LIN {X 0,Y 389.575,Z 385.776,A -85,B 0,C 180,E1 17407.486,E2 17407.486} C_VEL
LIN {X 0,Y 384.372,Z 564.348,A -85,B 0,C 180,E1 17404.221,E2 17404.221} C_VEL
LIN {X 0,Y 383.473,Z 583.113,A -85,B 0,C 180,E1 17403.623,E2 17403.623} C_VEL
LIN {X 0,Y 382.001,Z 600.901,A -85,B 0,C 180,E1 17402.806,E2 17402.806} C_VEL
LIN {X 0,Y 380.036,Z 618.183,A -85,B 0,C 180,E1 17401.748,E2 17401.748} C_VEL
LIN {X 0,Y 377.634,Z 634.674,A -85,B 0,C 180,E1 17400.465,E2 17400.465} C_VEL
LIN {X 0,Y 374.767,Z 651.083,A -85,B 0,C 180,E1 17398.874,E2 17398.874} C_VEL
LIN {X 0,Y 371.677,Z 666.384,A -85,B 0,C 180,E1 17397.04,E2 17397.04} C_VEL
LIN {X 0,Y 368.609,Z 680.089,A -85,B 0,C 180,E1 17395.033,E2 17395.033} C_VEL
LIN {X 0,Y 365.431,Z 693.192,A -85,B 0,C 180,E1 17392.692,E2 17392.692} C_VEL
LIN {X 0,Y 362.5,Z 704.69,A -85,B 0,C 180,E1 17390.168,E2 17390.168} C_VEL
LIN {X 0,Y 359.935,Z 714.65,A -85,B 0,C 180,E1 17387.458,E2 17387.458} C_VEL
LIN {X 0,Y 357.763,Z 723.094,A -85,B 0,C 180,E1 17384.568,E2 17384.568} C_VEL
LIN {X 0,Y 356.161,Z 729.667,A -85,B 0,C 180,E1 17381.661,E2 17381.661} C_VEL
LIN {X 0,Y 355.001,Z 734.817,A -85,B 0,C 180,E1 17378.585,E2 17378.585} C_VEL
LIN {X 0,Y 354.248,Z 738.439,A -85,B 0,C 180,E1 17375.344,E2 17375.344} C_VEL
LIN {X 0,Y 353.897,Z 740.346,A -85,B 0,C 180,E1 17372.105,E2 17372.105} C_VEL
LIN {X 0,Y 353.848,Z 740.616,A -85,B 0,C 180,E1 17368.867,E2 17368.867} C_VEL
LIN {X 0,Y 353.866,Z 740.566,A -85,B 0,C 180,E1 17368.451,E2 17368.451} C_VEL
LIN {X 0,Y 352.976,Z 740.398,A -85,B 0,C 180,E1 17367.201,E2 17367.201} C_VEL
LIN {X 0,Y 348.515,Z 739.641,A -85,B 0,C 180,E1 17364.746,E2 17364.746} C_VEL
LIN {X 0,Y 346.754,Z 738.536,A -85,B 0,C 180,E1 17363.218,E2 17363.218} C_VEL
LIN {X 0,Y 346.714,Z 738.05,A -85,B 0,C 180,E1 17362.764,E2 17362.764} C_VEL
LIN {X 0,Y 347.737,Z 733.66,A -85,B 0,C 180,E1 17359.537,E2 17359.537} C_VEL
LIN {X 0,Y 349.321,Z 727.307,A -85,B 0,C 180,E1 17356.257,E2 17356.257} C_VEL
LIN {X 0,Y 351.36,Z 719.697,A -85,B 0,C 180,E1 17353.297,E2 17353.297} C_VEL
LIN {X 0,Y 353.982,Z 710.063,A -85,B 0,C 180,E1 17350.36,E2 17350.36} C_VEL
LIN {X 0,Y 356.844,Z 699.482,A -85,B 0,C 180,E1 17347.775,E2 17347.775} C_VEL
LIN {X 0,Y 359.992,Z 687.464,A -85,B 0,C 180,E1 17345.38,E2 17345.38} C_VEL
LIN {X 0,Y 363.293,Z 673.927,A -85,B 0,C 180,E1 17343.17,E2 17343.17} C_VEL
LIN {X 0,Y 366.539,Z 659.329,A -85,B 0,C 180,E1 17341.22,E2 17341.22} C_VEL
LIN {X 0,Y 369.603,Z 643.731,A -85,B 0,C 180,E1 17339.522,E2 17339.522} C_VEL
LIN {X 0,Y 372.443,Z 626.719,A -85,B 0,C 180,E1 17338.031,E2 17338.031} C_VEL
LIN {X 0,Y 374.739,Z 609.542,A -85,B 0,C 180,E1 17336.842,E2 17336.842} C_VEL
LIN {X 0,Y 376.605,Z 590.744,A -85,B 0,C 180,E1 17335.852,E2 17335.852} C_VEL
LIN {X 0,Y 377.824,Z 571.243,A -85,B 0,C 180,E1 17335.127,E2 17335.127} C_VEL
LIN {X 0,Y 378.505,Z 547.045,A -85,B 0,C 180,E1 17334.58,E2 17334.58} C_VEL
LIN {X 0,Y 383.388,Z 388.518,A -85,B 0,C 180,E1 17331.66,E2 17331.66} C_VEL
LIN {X 0,Y 372.23,Z 368.985,A -85,B 0,C 180,E1 17329.629,E2 17329.629} C_VEL
LIN {X 0,Y 361.52,Z 352.259,A -85,B 0,C 180,E1 17327.541,E2 17327.541} C_VEL
LIN {X 0,Y 358.785,Z 347.938,A -85,B 0,C 180,E1 17326.899,E2 17326.899} C_VEL
LIN {X 0,Y 353.532,Z 335.825,A -85,B 0,C 180,E1 17323.861,E2 17323.861} C_VEL
LIN {X 0,Y 349.647,Z 327.602,A -85,B 0,C 180,E1 17321.563,E2 17321.563} C_VEL
LIN {X 0,Y 347.304,Z 322.978,A -85,B 0,C 180,E1 17320.157,E2 17320.157} C_VEL
LIN {X 0,Y 345.919,Z 319.541,A -85,B 0,C 180,E1 17319.059,E2 17319.059} C_VEL
LIN {X 0,Y 345.894,Z 319.384,A -85,B 0,C 180,E1 17314.823,E2 17314.823} C_VEL
LIN {X 0,Y 345.892,Z 319.382,A -85,B 0,C 180,E1 17310.527,E2 17310.527} C_VEL
LIN {X 0,Y 345.896,Z 319.388,A -85,B 0,C 180,E1 17306.354,E2 17306.354} C_VEL
LIN {X 0,Y 345.893,Z 319.4,A -85,B 0,C 180,E1 17302.252,E2 17302.252} C_VEL
LIN {X 0,Y 345.899,Z 319.385,A -85,B 0,C 180,E1 17298.014,E2 17298.014} C_VEL
LIN {X 0,Y 345.906,Z 319.366,A -85,B 0,C 180,E1 17293.785,E2 17293.785} C_VEL
LIN {X 0,Y 345.898,Z 319.37,A -85,B 0,C 180,E1 17289.484,E2 17289.484} C_VEL
LIN {X 0,Y 345.89,Z 319.398,A -85,B 0,C 180,E1 17285.308,E2 17285.308} C_VEL
LIN {X 0,Y 345.877,Z 319.386,A -85,B 0,C 180,E1 17281.16,E2 17281.16} C_VEL
LIN {X 0,Y 345.871,Z 319.369,A -85,B 0,C 180,E1 17277.018,E2 17277.018} C_VEL
LIN {X 0,Y 345.87,Z 319.378,A -85,B 0,C 180,E1 17272.86,E2 17272.86} C_VEL
LIN {X 0,Y 345.873,Z 319.401,A -85,B 0,C 180,E1 17268.664,E2 17268.664} C_VEL
LIN {X 0,Y 345.873,Z 319.4,A -85,B 0,C 180,E1 17264.405,E2 17264.405} C_VEL
LIN {X 0,Y 345.88,Z 319.39,A -85,B 0,C 180,E1 17260.056,E2 17260.056} C_VEL
LIN {X 0,Y 345.886,Z 319.384,A -85,B 0,C 180,E1 17255.947,E2 17255.947} C_VEL
LIN {X 0,Y 345.901,Z 319.385,A -85,B 0,C 180,E1 17251.702,E2 17251.702} C_VEL
LIN {X 0,Y 345.947,Z 319.628,A -85,B 0,C 180,E1 17249.507,E2 17249.507} C_VEL
LIN {X 0,Y 347.584,Z 323.392,A -85,B 0,C 180,E1 17248.43,E2 17248.43} C_VEL
LIN {X 0,Y 348.628,Z 324.913,A -85,B 0,C 180,E1 17247.956,E2 17247.956} C_VEL
LIN {X 0,Y 353.831,Z 334.918,A -85,B 0,C 180,E1 17245.39,E2 17245.39} C_VEL
LIN {X 0,Y 357.949,Z 342.981,A -85,B 0,C 180,E1 17243.49,E2 17243.49} C_VEL
LIN {X 0,Y 364.694,Z 357.152,A -85,B 0,C 180,E1 17240.502,E2 17240.502} C_VEL
LIN {X 0,Y 371.956,Z 374.258,A -85,B 0,C 180,E1 17237.359,E2 17237.359} C_VEL
LIN {X 0,Y 374.056,Z 379.335,A -85,B 0,C 180,E1 17236.557,E2 17236.557} C_VEL
LIN {X 0,Y 381.034,Z 392.431,A -85,B 0,C 180,E1 17235.246,E2 17235.246} C_VEL
LIN {X 0,Y 383.985,Z 429.126,A -85,B 0,C 180,E1 17233.918,E2 17233.918} C_VEL
LIN {X 0,Y 375.667,Z 632.493,A -85,B 0,C 180,E1 17229.71,E2 17229.71} C_VEL
LIN {X 0,Y 373.709,Z 654.478,A -85,B 0,C 180,E1 17229.004,E2 17229.004} C_VEL
LIN {X 0,Y 371.041,Z 675.386,A -85,B 0,C 180,E1 17228.054,E2 17228.054} C_VEL
LIN {X 0,Y 368.083,Z 694.62,A -85,B 0,C 180,E1 17226.892,E2 17226.892} C_VEL
LIN {X 0,Y 364.802,Z 713.742,A -85,B 0,C 180,E1 17225.427,E2 17225.427} C_VEL
LIN {X 0,Y 361.389,Z 732.08,A -85,B 0,C 180,E1 17223.691,E2 17223.691} C_VEL
LIN {X 0,Y 357.817,Z 750.227,A -85,B 0,C 180,E1 17221.596,E2 17221.596} C_VEL
LIN {X 0,Y 354.467,Z 767.276,A -85,B 0,C 180,E1 17219.207,E2 17219.207} C_VEL
LIN {X 0,Y 351.414,Z 783.149,A -85,B 0,C 180,E1 17216.531,E2 17216.531} C_VEL
LIN {X 0,Y 348.903,Z 797.366,A -85,B 0,C 180,E1 17213.653,E2 17213.653} C_VEL
LIN {X 0,Y 346.99,Z 809.978,A -85,B 0,C 180,E1 17210.581,E2 17210.581} C_VEL
LIN {X 0,Y 345.729,Z 820.44,A -85,B 0,C 180,E1 17207.503,E2 17207.503} C_VEL
LIN {X 0,Y 345.044,Z 829.017,A -85,B 0,C 180,E1 17204.43,E2 17204.43} C_VEL
LIN {X 0,Y 344.787,Z 836.104,A -85,B 0,C 180,E1 17201.203,E2 17201.203} C_VEL
LIN {X 0,Y 344.85,Z 841.123,A -85,B 0,C 180,E1 17198.167,E2 17198.167} C_VEL
LIN {X 0,Y 345.058,Z 844.743,A -85,B 0,C 180,E1 17194.987,E2 17194.987} C_VEL
LIN {X 0,Y 345.211,Z 846.508,A -85,B 0,C 180,E1 17192.158,E2 17192.158} C_VEL
LIN {X 0,Y 345.255,Z 846.827,A -85,B 0,C 180,E1 17189.17,E2 17189.17} C_VEL
LIN {X 0,Y 345.126,Z 845.656,A -85,B 0,C 180,E1 17186.179,E2 17186.179} C_VEL
LIN {X 0,Y 344.931,Z 842.863,A -85,B 0,C 180,E1 17183.175,E2 17183.175} C_VEL
LIN {X 0,Y 344.793,Z 838.223,A -85,B 0,C 180,E1 17179.98,E2 17179.98} C_VEL
LIN {X 0,Y 344.896,Z 831.799,A -85,B 0,C 180,E1 17176.761,E2 17176.761} C_VEL
LIN {X 0,Y 345.408,Z 823.997,A -85,B 0,C 180,E1 17173.693,E2 17173.693} C_VEL
LIN {X 0,Y 346.494,Z 813.722,A -85,B 0,C 180,E1 17170.444,E2 17170.444} C_VEL
LIN {X 0,Y 348.173,Z 801.841,A -85,B 0,C 180,E1 17167.369,E2 17167.369} C_VEL
LIN {X 0,Y 350.447,Z 788.441,A -85,B 0,C 180,E1 17164.481,E2 17164.481} C_VEL
LIN {X 0,Y 353.14,Z 774.009,A -85,B 0,C 180,E1 17161.874,E2 17161.874} C_VEL
LIN {X 0,Y 356.244,Z 758.161,A -85,B 0,C 180,E1 17159.47,E2 17159.47} C_VEL
LIN {X 0,Y 359.673,Z 740.767,A -85,B 0,C 180,E1 17157.27,E2 17157.27} C_VEL
LIN {X 0,Y 363.194,Z 722.371,A -85,B 0,C 180,E1 17155.356,E2 17155.356} C_VEL
LIN {X 0,Y 366.647,Z 702.966,A -85,B 0,C 180,E1 17153.719,E2 17153.719} C_VEL
LIN {X 0,Y 369.743,Z 683.735,A -85,B 0,C 180,E1 17152.426,E2 17152.426} C_VEL
LIN {X 0,Y 372.564,Z 663.659,A -85,B 0,C 180,E1 17151.389,E2 17151.389} C_VEL
LIN {X 0,Y 374.836,Z 642.783,A -85,B 0,C 180,E1 17150.598,E2 17150.598} C_VEL
LIN {X 0,Y 376.217,Z 620.758,A -85,B 0,C 180,E1 17150.027,E2 17150.027} C_VEL
LIN {X 0,Y 383.944,Z 427.198,A -85,B 0,C 180,E1 17146.047,E2 17146.047} C_VEL
LIN {X 0,Y 380.702,Z 391.532,A -85,B 0,C 180,E1 17144.711,E2 17144.711} C_VEL
LIN {X 0,Y 373.38,Z 377.914,A -85,B 0,C 180,E1 17143.277,E2 17143.277} C_VEL
LIN {X 0,Y 366.854,Z 362.006,A -85,B 0,C 180,E1 17140.441,E2 17140.441} C_VEL
LIN {X 0,Y 360.67,Z 348.666,A -85,B 0,C 180,E1 17137.782,E2 17137.782} C_VEL
LIN {X 0,Y 355.146,Z 337.373,A -85,B 0,C 180,E1 17135.25,E2 17135.25} C_VEL
LIN {X 0,Y 350.284,Z 328.233,A -85,B 0,C 180,E1 17132.947,E2 17132.947} C_VEL
LIN {X 0,Y 348.264,Z 324.159,A -85,B 0,C 180,E1 17131.888,E2 17131.888} C_VEL
LIN {X 0,Y 346.287,Z 320.952,A -85,B 0,C 180,E1 17130.927,E2 17130.927} C_VEL
LIN {X 0,Y 345.918,Z 319.456,A -85,B 0,C 180,E1 17130.413,E2 17130.413} C_VEL
LIN {X 0,Y 345.898,Z 319.385,A -85,B 0,C 180,E1 17126.248,E2 17126.248} C_VEL
LIN {X 0,Y 345.886,Z 319.383,A -85,B 0,C 180,E1 17122.073,E2 17122.073} C_VEL
LIN {X 0,Y 345.877,Z 319.378,A -85,B 0,C 180,E1 17117.844,E2 17117.844} C_VEL
LIN {X 0,Y 345.87,Z 319.372,A -85,B 0,C 180,E1 17113.542,E2 17113.542} C_VEL
LIN {X 0,Y 345.87,Z 319.379,A -85,B 0,C 180,E1 17109.316,E2 17109.316} C_VEL
LIN {X 0,Y 345.873,Z 319.402,A -85,B 0,C 180,E1 17105.141,E2 17105.141} C_VEL
LIN {X 0,Y 345.872,Z 319.39,A -85,B 0,C 180,E1 17100.993,E2 17100.993} C_VEL
LIN {X 0,Y 345.87,Z 319.369,A -85,B 0,C 180,E1 17096.851,E2 17096.851} C_VEL
LIN {X 0,Y 345.884,Z 319.379,A -85,B 0,C 180,E1 17092.692,E2 17092.692} C_VEL
LIN {X 0,Y 345.897,Z 319.401,A -85,B 0,C 180,E1 17088.491,E2 17088.491} C_VEL
LIN {X 0,Y 345.908,Z 319.379,A -85,B 0,C 180,E1 17084.234,E2 17084.234} C_VEL
LIN {X 0,Y 345.896,Z 319.37,A -85,B 0,C 180,E1 17079.956,E2 17079.956} C_VEL
LIN {X 0,Y 345.902,Z 319.373,A -85,B 0,C 180,E1 17075.947,E2 17075.947} C_VEL
LIN {X 0,Y 345.896,Z 319.385,A -85,B 0,C 180,E1 17071.701,E2 17071.701} C_VEL
LIN {X 0,Y 345.897,Z 319.393,A -85,B 0,C 180,E1 17067.569,E2 17067.569} C_VEL
LIN {X 0,Y 345.896,Z 319.393,A -85,B 0,C 180,E1 17063.453,E2 17063.453} C_VEL
LIN {X 0,Y 345.937,Z 319.68,A -85,B 0,C 180,E1 17060.73,E2 17060.73} C_VEL
LIN {X 0,Y 347.422,Z 323.162,A -85,B 0,C 180,E1 17059.643,E2 17059.643} C_VEL
LIN {X 0,Y 348.545,Z 325.55,A -85,B 0,C 180,E1 17058.934,E2 17058.934} C_VEL
LIN {X 0,Y 350.596,Z 329.771,A -85,B 0,C 180,E1 17057.697,E2 17057.697} C_VEL
LIN {X 0,Y 354.243,Z 337.521,A -85,B 0,C 180,E1 17055.568,E2 17055.568} C_VEL
LIN {X 0,Y 358.954,Z 348.373,A -85,B 0,C 180,E1 17052.896,E2 17052.896} C_VEL
LIN {X 0,Y 369.652,Z 364.898,A -85,B 0,C 180,E1 17050.738,E2 17050.738} C_VEL
LIN {X 0,Y 379.94,Z 382.361,A -85,B 0,C 180,E1 17048.834,E2 17048.834} C_VEL
LIN {X 0,Y 383.444,Z 389.074,A -85,B 0,C 180,E1 17048.206,E2 17048.206} C_VEL
LIN {X 0,Y 378.018,Z 564.942,A -85,B 0,C 180,E1 17044.946,E2 17044.946} C_VEL
LIN {X 0,Y 377.086,Z 583.644,A -85,B 0,C 180,E1 17044.345,E2 17044.345} C_VEL
LIN {X 0,Y 375.513,Z 601.927,A -85,B 0,C 180,E1 17043.496,E2 17043.496} C_VEL
LIN {X 0,Y 373.525,Z 618.693,A -85,B 0,C 180,E1 17042.458,E2 17042.458} C_VEL
LIN {X 0,Y 370.899,Z 636.019,A -85,B 0,C 180,E1 17041.094,E2 17041.094} C_VEL
LIN {X 0,Y 367.89,Z 652.482,A -85,B 0,C 180,E1 17039.466,E2 17039.466} C_VEL
LIN {X 0,Y 364.669,Z 667.723,A -85,B 0,C 180,E1 17037.604,E2 17037.604} C_VEL
LIN {X 0,Y 361.466,Z 681.388,A -85,B 0,C 180,E1 17035.563,E2 17035.563} C_VEL
LIN {X 0,Y 358.145,Z 694.464,A -85,B 0,C 180,E1 17033.18,E2 17033.18} C_VEL
LIN {X 0,Y 355.074,Z 705.939,A -85,B 0,C 180,E1 17030.608,E2 17030.608} C_VEL
LIN {X 0,Y 352.38,Z 715.885,A -85,B 0,C 180,E1 17027.845,E2 17027.845} C_VEL
LIN {X 0,Y 350.093,Z 724.318,A -85,B 0,C 180,E1 17024.894,E2 17024.894} C_VEL
LIN {X 0,Y 348.354,Z 731.066,A -85,B 0,C 180,E1 17021.831,E2 17021.831} C_VEL
LIN {X 0,Y 347.117,Z 736.256,A -85,B 0,C 180,E1 17018.614,E2 17018.614} C_VEL
LIN {X 0,Y 346.367,Z 739.644,A -85,B 0,C 180,E1 17015.466,E2 17015.466} C_VEL
LIN {X 0,Y 345.992,Z 741.548,A -85,B 0,C 180,E1 17012.153,E2 17012.153} C_VEL
LIN {X 0,Y 345.939,Z 741.818,A -85,B 0,C 180,E1 17008.841,E2 17008.841} C_VEL
LIN {X 0,Y 346.204,Z 740.465,A -85,B 0,C 180,E1 17005.528,E2 17005.528} C_VEL
LIN {X 0,Y 346.714,Z 738.05,A -85,B 0,C 180,E1 17002.764,E2 17002.764} C_VEL
LIN {X 0,Y 346.061,Z 736.752,A -85,B 0,C 180,E1 17001.504,E2 17001.504} C_VEL
LIN {X 0,Y 341.253,Z 732.89,A -85,B 0,C 180,E1 16998.207,E2 16998.207} C_VEL
LIN {X 0,Y 340.994,Z 730.849,A -85,B 0,C 180,E1 16997.039,E2 16997.039} C_VEL
LIN {X 0,Y 342.986,Z 723.691,A -85,B 0,C 180,E1 16993.923,E2 16993.923} C_VEL
LIN {X 0,Y 345.546,Z 714.785,A -85,B 0,C 180,E1 16990.916,E2 16990.916} C_VEL
LIN {X 0,Y 348.539,Z 704.306,A -85,B 0,C 180,E1 16988.104,E2 16988.104} C_VEL
LIN {X 0,Y 351.909,Z 692.224,A -85,B 0,C 180,E1 16985.493,E2 16985.493} C_VEL
LIN {X 0,Y 355.499,Z 678.411,A -85,B 0,C 180,E1 16983.076,E2 16983.076} C_VEL
LIN {X 0,Y 358.999,Z 663.723,A -85,B 0,C 180,E1 16980.99,E2 16980.99} C_VEL
LIN {X 0,Y 362.256,Z 648.294,A -85,B 0,C 180,E1 16979.204,E2 16979.204} C_VEL
LIN {X 0,Y 365.281,Z 631.623,A -85,B 0,C 180,E1 16977.648,E2 16977.648} C_VEL
LIN {X 0,Y 367.892,Z 613.759,A -85,B 0,C 180,E1 16976.33,E2 16976.33} C_VEL
LIN {X 0,Y 369.927,Z 595.416,A -85,B 0,C 180,E1 16975.295,E2 16975.295} C_VEL
LIN {X 0,Y 371.317,Z 576.435,A -85,B 0,C 180,E1 16974.519,E2 16974.519} C_VEL
LIN {X 0,Y 372.031,Z 556.598,A -85,B 0,C 180,E1 16973.998,E2 16973.998} C_VEL
LIN {X 0,Y 377.33,Z 391.658,A -85,B 0,C 180,E1 16970.912,E2 16970.912} C_VEL
LIN {X 0,Y 366.892,Z 373.263,A -85,B 0,C 180,E1 16968.936,E2 16968.936} C_VEL
LIN {X 0,Y 356.62,Z 357.168,A -85,B 0,C 180,E1 16966.859,E2 16966.859} C_VEL
LIN {X 0,Y 351.137,Z 348.844,A -85,B 0,C 180,E1 16965.621,E2 16965.621} C_VEL
LIN {X 0,Y 345.873,Z 337.173,A -85,B 0,C 180,E1 16962.512,E2 16962.512} C_VEL
LIN {X 0,Y 341.765,Z 328.63,A -85,B 0,C 180,E1 16959.961,E2 16959.961} C_VEL
LIN {X 0,Y 339.688,Z 324.424,A -85,B 0,C 180,E1 16958.61,E2 16958.61} C_VEL
LIN {X 0,Y 337.986,Z 320.54,A -85,B 0,C 180,E1 16957.273,E2 16957.273} C_VEL
LIN {X 0,Y 337.951,Z 320.371,A -85,B 0,C 180,E1 16952.983,E2 16952.983} C_VEL
LIN {X 0,Y 337.95,Z 320.368,A -85,B 0,C 180,E1 16948.64,E2 16948.64} C_VEL
LIN {X 0,Y 337.952,Z 320.361,A -85,B 0,C 180,E1 16944.326,E2 16944.326} C_VEL
LIN {X 0,Y 337.949,Z 320.361,A -85,B 0,C 180,E1 16940.253,E2 16940.253} C_VEL
LIN {X 0,Y 337.96,Z 320.373,A -85,B 0,C 180,E1 16935.953,E2 16935.953} C_VEL
LIN {X 0,Y 337.964,Z 320.385,A -85,B 0,C 180,E1 16931.699,E2 16931.699} C_VEL
LIN {X 0,Y 337.964,Z 320.361,A -85,B 0,C 180,E1 16927.48,E2 16927.48} C_VEL
LIN {X 0,Y 337.939,Z 320.356,A -85,B 0,C 180,E1 16923.223,E2 16923.223} C_VEL
LIN {X 0,Y 337.929,Z 320.376,A -85,B 0,C 180,E1 16918.983,E2 16918.983} C_VEL
LIN {X 0,Y 337.927,Z 320.39,A -85,B 0,C 180,E1 16914.738,E2 16914.738} C_VEL
LIN {X 0,Y 337.926,Z 320.37,A -85,B 0,C 180,E1 16910.463,E2 16910.463} C_VEL
LIN {X 0,Y 337.932,Z 320.361,A -85,B 0,C 180,E1 16906.134,E2 16906.134} C_VEL
LIN {X 0,Y 337.943,Z 320.364,A -85,B 0,C 180,E1 16901.901,E2 16901.901} C_VEL
LIN {X 0,Y 337.955,Z 320.368,A -85,B 0,C 180,E1 16897.748,E2 16897.748} C_VEL
LIN {X 0,Y 337.969,Z 320.367,A -85,B 0,C 180,E1 16893.467,E2 16893.467} C_VEL
LIN {X 0,Y 338.026,Z 320.649,A -85,B 0,C 180,E1 16891.307,E2 16891.307} C_VEL
LIN {X 0,Y 339.317,Z 323.956,A -85,B 0,C 180,E1 16890.328,E2 16890.328} C_VEL
LIN {X 0,Y 340.859,Z 326.12,A -85,B 0,C 180,E1 16889.585,E2 16889.585} C_VEL
LIN {X 0,Y 342.798,Z 329.791,A -85,B 0,C 180,E1 16888.527,E2 16888.527} C_VEL
LIN {X 0,Y 348.279,Z 340.218,A -85,B 0,C 180,E1 16885.758,E2 16885.758} C_VEL
LIN {X 0,Y 354.382,Z 352.579,A -85,B 0,C 180,E1 16882.859,E2 16882.859} C_VEL
LIN {X 0,Y 360.708,Z 366.49,A -85,B 0,C 180,E1 16879.978,E2 16879.978} C_VEL
LIN {X 0,Y 365.81,Z 378.592,A -85,B 0,C 180,E1 16877.802,E2 16877.802} C_VEL
LIN {X 0,Y 375.242,Z 395.721,A -85,B 0,C 180,E1 16875.957,E2 16875.957} C_VEL
LIN {X 0,Y 377.885,Z 430.233,A -85,B 0,C 180,E1 16874.686,E2 16874.686} C_VEL
LIN {X 0,Y 369.297,Z 631.618,A -85,B 0,C 180,E1 16870.468,E2 16870.468} C_VEL
LIN {X 0,Y 367.272,Z 653.63,A -85,B 0,C 180,E1 16869.753,E2 16869.753} C_VEL
LIN {X 0,Y 364.435,Z 674.971,A -85,B 0,C 180,E1 16868.771,E2 16868.771} C_VEL
LIN {X 0,Y 361.176,Z 695.239,A -85,B 0,C 180,E1 16867.518,E2 16867.518} C_VEL
LIN {X 0,Y 357.602,Z 714.966,A -85,B 0,C 180,E1 16865.955,E2 16865.955} C_VEL
LIN {X 0,Y 353.991,Z 733.289,A -85,B 0,C 180,E1 16864.149,E2 16864.149} C_VEL
LIN {X 0,Y 350.491,Z 750.079,A -85,B 0,C 180,E1 16862.142,E2 16862.142} C_VEL
LIN {X 0,Y 347.071,Z 766.57,A -85,B 0,C 180,E1 16859.772,E2 16859.772} C_VEL
LIN {X 0,Y 343.961,Z 781.792,A -85,B 0,C 180,E1 16857.153,E2 16857.153} C_VEL
LIN {X 0,Y 341.276,Z 796.036,A -85,B 0,C 180,E1 16854.215,E2 16854.215} C_VEL
LIN {X 0,Y 339.307,Z 808.039,A -85,B 0,C 180,E1 16851.25,E2 16851.25} C_VEL
LIN {X 0,Y 337.908,Z 818.643,A -85,B 0,C 180,E1 16848.1,E2 16848.1} C_VEL
LIN {X 0,Y 337.111,Z 827.752,A -85,B 0,C 180,E1 16844.777,E2 16844.777} C_VEL
LIN {X 0,Y 336.824,Z 834.857,A -85,B 0,C 180,E1 16841.472,E2 16841.472} C_VEL
LIN {X 0,Y 336.893,Z 839.896,A -85,B 0,C 180,E1 16838.362,E2 16838.362} C_VEL
LIN {X 0,Y 337.125,Z 843.531,A -85,B 0,C 180,E1 16835.104,E2 16835.104} C_VEL
LIN {X 0,Y 337.296,Z 845.304,A -85,B 0,C 180,E1 16832.208,E2 16832.208} C_VEL
LIN {X 0,Y 337.344,Z 845.625,A -85,B 0,C 180,E1 16829.151,E2 16829.151} C_VEL
LIN {X 0,Y 337.2,Z 844.447,A -85,B 0,C 180,E1 16826.09,E2 16826.09} C_VEL
LIN {X 0,Y 336.979,Z 841.641,A -85,B 0,C 180,E1 16823.013,E2 16823.013} C_VEL
LIN {X 0,Y 336.832,Z 836.984,A -85,B 0,C 180,E1 16819.741,E2 16819.741} C_VEL
LIN {X 0,Y 336.947,Z 830.538,A -85,B 0,C 180,E1 16816.443,E2 16816.443} C_VEL
LIN {X 0,Y 337.497,Z 822.711,A -85,B 0,C 180,E1 16813.3,E2 16813.3} C_VEL
LIN {X 0,Y 338.683,Z 812.419,A -85,B 0,C 180,E1 16809.974,E2 16809.974} C_VEL
LIN {X 0,Y 340.528,Z 800.34,A -85,B 0,C 180,E1 16806.784,E2 16806.784} C_VEL
LIN {X 0,Y 342.929,Z 787.093,A -85,B 0,C 180,E1 16803.88,E2 16803.88} C_VEL
LIN {X 0,Y 345.7,Z 773.129,A -85,B 0,C 180,E1 16801.308,E2 16801.308} C_VEL
LIN {X 0,Y 348.97,Z 757.336,A -85,B 0,C 180,E1 16798.859,E2 16798.859} C_VEL
LIN {X 0,Y 352.569,Z 740.004,A -85,B 0,C 180,E1 16796.622,E2 16796.622} C_VEL
LIN {X 0,Y 356.261,Z 721.682,A -85,B 0,C 180,E1 16794.681,E2 16794.681} C_VEL
LIN {X 0,Y 359.684,Z 703.397,A -85,B 0,C 180,E1 16793.1,E2 16793.1} C_VEL
LIN {X 0,Y 362.893,Z 684.551,A -85,B 0,C 180,E1 16791.791,E2 16791.791} C_VEL
LIN {X 0,Y 365.952,Z 663.876,A -85,B 0,C 180,E1 16790.69,E2 16790.69} C_VEL
LIN {X 0,Y 368.407,Z 642.256,A -85,B 0,C 180,E1 16789.855,E2 16789.855} C_VEL
LIN {X 0,Y 369.854,Z 620.163,A -85,B 0,C 180,E1 16789.272,E2 16789.272} C_VEL
LIN {X 0,Y 377.84,Z 428.2,A -85,B 0,C 180,E1 16785.277,E2 16785.277} C_VEL
LIN {X 0,Y 374.987,Z 395.198,A -85,B 0,C 180,E1 16784.021,E2 16784.021} C_VEL
LIN {X 0,Y 365.339,Z 377.727,A -85,B 0,C 180,E1 16782.106,E2 16782.106} C_VEL
LIN {X 0,Y 358.592,Z 361.64,A -85,B 0,C 180,E1 16779.061,E2 16779.061} C_VEL
LIN {X 0,Y 351.937,Z 347.377,A -85,B 0,C 180,E1 16776.021,E2 16776.021} C_VEL
LIN {X 0,Y 346.773,Z 337.483,A -85,B 0,C 180,E1 16773.565,E2 16773.565} C_VEL
LIN {X 0,Y 344.569,Z 333.342,A -85,B 0,C 180,E1 16772.468,E2 16772.468} C_VEL
LIN {X 0,Y 342.71,Z 329.695,A -85,B 0,C 180,E1 16771.482,E2 16771.482} C_VEL
LIN {X 0,Y 340.761,Z 325.802,A -85,B 0,C 180,E1 16770.387,E2 16770.387} C_VEL
LIN {X 0,Y 338.388,Z 322.126,A -85,B 0,C 180,E1 16769.178,E2 16769.178} C_VEL
LIN {X 0,Y 338,Z 320.488,A -85,B 0,C 180,E1 16768.634,E2 16768.634} C_VEL
LIN {X 0,Y 337.962,Z 320.376,A -85,B 0,C 180,E1 16764.33,E2 16764.33} C_VEL
LIN {X 0,Y 337.957,Z 320.383,A -85,B 0,C 180,E1 16760.252,E2 16760.252} C_VEL
LIN {X 0,Y 337.942,Z 320.391,A -85,B 0,C 180,E1 16755.942,E2 16755.942} C_VEL
LIN {X 0,Y 337.932,Z 320.383,A -85,B 0,C 180,E1 16751.607,E2 16751.607} C_VEL
LIN {X 0,Y 337.928,Z 320.366,A -85,B 0,C 180,E1 16747.309,E2 16747.309} C_VEL
LIN {X 0,Y 337.93,Z 320.359,A -85,B 0,C 180,E1 16743.053,E2 16743.053} C_VEL
LIN {X 0,Y 337.931,Z 320.38,A -85,B 0,C 180,E1 16738.982,E2 16738.982} C_VEL
LIN {X 0,Y 337.943,Z 320.386,A -85,B 0,C 180,E1 16734.737,E2 16734.737} C_VEL
LIN {X 0,Y 337.954,Z 320.359,A -85,B 0,C 180,E1 16730.463,E2 16730.463} C_VEL
LIN {X 0,Y 337.957,Z 320.356,A -85,B 0,C 180,E1 16726.134,E2 16726.134} C_VEL
LIN {X 0,Y 337.951,Z 320.374,A -85,B 0,C 180,E1 16721.901,E2 16721.901} C_VEL
LIN {X 0,Y 337.951,Z 320.389,A -85,B 0,C 180,E1 16717.746,E2 16717.746} C_VEL
LIN {X 0,Y 337.946,Z 320.38,A -85,B 0,C 180,E1 16713.464,E2 16713.464} C_VEL
LIN {X 0,Y 337.945,Z 320.375,A -85,B 0,C 180,E1 16709.213,E2 16709.213} C_VEL
LIN {X 0,Y 337.949,Z 320.375,A -85,B 0,C 180,E1 16704.972,E2 16704.972} C_VEL
LIN {X 0,Y 338.009,Z 320.663,A -85,B 0,C 180,E1 16702.511,E2 16702.511} C_VEL
LIN {X 0,Y 339.793,Z 324.568,A -85,B 0,C 180,E1 16701.188,E2 16701.188} C_VEL
LIN {X 0,Y 342.825,Z 330.891,A -85,B 0,C 180,E1 16699.208,E2 16699.208} C_VEL
LIN {X 0,Y 346.651,Z 338.868,A -85,B 0,C 180,E1 16696.875,E2 16696.875} C_VEL
LIN {X 0,Y 351.508,Z 349.594,A -85,B 0,C 180,E1 16694.12,E2 16694.12} C_VEL
LIN {X 0,Y 362.352,Z 366.047,A -85,B 0,C 180,E1 16691.838,E2 16691.838} C_VEL
LIN {X 0,Y 373.097,Z 384.003,A -85,B 0,C 180,E1 16689.754,E2 16689.754} C_VEL
LIN {X 0,Y 377.371,Z 392.19,A -85,B 0,C 180,E1 16688.955,E2 16688.955} C_VEL
LIN {X 0,Y 371.728,Z 565.463,A -85,B 0,C 180,E1 16685.698,E2 16685.698} C_VEL
LIN {X 0,Y 370.761,Z 584.169,A -85,B 0,C 180,E1 16685.093,E2 16685.093} C_VEL
LIN {X 0,Y 369.14,Z 602.364,A -85,B 0,C 180,E1 16684.243,E2 16684.243} C_VEL
LIN {X 0,Y 366.924,Z 620.305,A -85,B 0,C 180,E1 16683.116,E2 16683.116} C_VEL
LIN {X 0,Y 364.314,Z 636.765,A -85,B 0,C 180,E1 16681.798,E2 16681.798} C_VEL
LIN {X 0,Y 361.195,Z 653.169,A -85,B 0,C 180,E1 16680.16,E2 16680.16} C_VEL
LIN {X 0,Y 357.832,Z 668.479,A -85,B 0,C 180,E1 16678.269,E2 16678.269} C_VEL
LIN {X 0,Y 354.354,Z 682.686,A -85,B 0,C 180,E1 16676.114,E2 16676.114} C_VEL
LIN {X 0,Y 351.104,Z 694.934,A -85,B 0,C 180,E1 16673.852,E2 16673.852} C_VEL
LIN {X 0,Y 347.854,Z 706.532,A -85,B 0,C 180,E1 16671.233,E2 16671.233} C_VEL
LIN {X 0,Y 344.99,Z 716.587,A -85,B 0,C 180,E1 16668.415,E2 16668.415} C_VEL
LIN {X 0,Y 342.551,Z 725.119,A -85,B 0,C 180,E1 16665.403,E2 16665.403} C_VEL
LIN {X 0,Y 340.64,Z 732.111,A -85,B 0,C 180,E1 16662.194,E2 16662.194} C_VEL
LIN {X 0,Y 339.338,Z 737.236,A -85,B 0,C 180,E1 16658.984,E2 16658.984} C_VEL
LIN {X 0,Y 338.486,Z 740.849,A -85,B 0,C 180,E1 16655.594,E2 16655.594} C_VEL
LIN {X 0,Y 338.087,Z 742.75,A -85,B 0,C 180,E1 16652.203,E2 16652.203} C_VEL
LIN {X 0,Y 338.031,Z 743.019,A -85,B 0,C 180,E1 16648.814,E2 16648.814} C_VEL
LIN {X 0,Y 338.314,Z 741.668,A -85,B 0,C 180,E1 16645.423,E2 16645.423} C_VEL
LIN {X 0,Y 339.006,Z 738.638,A -85,B 0,C 180,E1 16642.032,E2 16642.032} C_VEL
LIN {X 0,Y 340.139,Z 734.091,A -85,B 0,C 180,E1 16638.813,E2 16638.813} C_VEL
LIN {X 0,Y 340.994,Z 730.849,A -85,B 0,C 180,E1 16637.039,E2 16637.039} C_VEL
LIN {X 0,Y 340.753,Z 728.553,A -85,B 0,C 180,E1 16635.793,E2 16635.793} C_VEL
LIN {X 0,Y 337.133,Z 722.237,A -85,B 0,C 180,E1 16632.617,E2 16632.617} C_VEL
LIN {X 0,Y 337.17,Z 718.967,A -85,B 0,C 180,E1 16631.419,E2 16631.419} C_VEL
LIN {X 0,Y 340.019,Z 709.487,A -85,B 0,C 180,E1 16628.616,E2 16628.616} C_VEL
LIN {X 0,Y 343.339,Z 698.274,A -85,B 0,C 180,E1 16625.94,E2 16625.94} C_VEL
LIN {X 0,Y 346.919,Z 685.521,A -85,B 0,C 180,E1 16623.467,E2 16623.467} C_VEL
LIN {X 0,Y 350.51,Z 671.669,A -85,B 0,C 180,E1 16621.272,E2 16621.272} C_VEL
LIN {X 0,Y 353.941,Z 657.099,A -85,B 0,C 180,E1 16619.382,E2 16619.382} C_VEL
LIN {X 0,Y 357.224,Z 641.016,A -85,B 0,C 180,E1 16617.684,E2 16617.684} C_VEL
LIN {X 0,Y 360.105,Z 624.301,A -85,B 0,C 180,E1 16616.269,E2 16616.269} C_VEL
LIN {X 0,Y 362.509,Z 606.576,A -85,B 0,C 180,E1 16615.089,E2 16615.089} C_VEL
LIN {X 0,Y 364.381,Z 587.477,A -85,B 0,C 180,E1 16614.139,E2 16614.139} C_VEL
LIN {X 0,Y 365.522,Z 567.969,A -85,B 0,C 180,E1 16613.47,E2 16613.47} C_VEL
LIN {X 0,Y 367.415,Z 507.805,A -85,B 0,C 180,E1 16612.286,E2 16612.286} C_VEL
LIN {X 0,Y 371.29,Z 394.593,A -85,B 0,C 180,E1 16610.129,E2 16610.129} C_VEL
LIN {X 0,Y 360.772,Z 376.206,A -85,B 0,C 180,E1 16608.055,E2 16608.055} C_VEL
LIN {X 0,Y 350.107,Z 359.514,A -85,B 0,C 180,E1 16605.793,E2 16605.793} C_VEL
LIN {X 0,Y 343.368,Z 349.702,A -85,B 0,C 180,E1 16604.22,E2 16604.22} C_VEL
LIN {X 0,Y 338.518,Z 338.884,A -85,B 0,C 180,E1 16601.198,E2 16601.198} C_VEL
LIN {X 0,Y 334.18,Z 330.098,A -85,B 0,C 180,E1 16598.383,E2 16598.383} C_VEL
LIN {X 0,Y 331.916,Z 325.62,A -85,B 0,C 180,E1 16596.832,E2 16596.832} C_VEL
LIN {X 0,Y 330.164,Z 322.103,A -85,B 0,C 180,E1 16595.553,E2 16595.553} C_VEL
LIN {X 0,Y 330.019,Z 321.371,A -85,B 0,C 180,E1 16594.933,E2 16594.933} C_VEL
LIN {X 0,Y 330.012,Z 321.359,A -85,B 0,C 180,E1 16590.598,E2 16590.598} C_VEL
LIN {X 0,Y 330.014,Z 321.367,A -85,B 0,C 180,E1 16586.448,E2 16586.448} C_VEL
LIN {X 0,Y 330.027,Z 321.377,A -85,B 0,C 180,E1 16582.066,E2 16582.066} C_VEL
LIN {X 0,Y 330.032,Z 321.367,A -85,B 0,C 180,E1 16577.636,E2 16577.636} C_VEL
LIN {X 0,Y 330.013,Z 321.348,A -85,B 0,C 180,E1 16573.313,E2 16573.313} C_VEL
LIN {X 0,Y 329.992,Z 321.345,A -85,B 0,C 180,E1 16568.984,E2 16568.984} C_VEL
LIN {X 0,Y 329.984,Z 321.366,A -85,B 0,C 180,E1 16564.693,E2 16564.693} C_VEL
LIN {X 0,Y 329.979,Z 321.379,A -85,B 0,C 180,E1 16560.348,E2 16560.348} C_VEL
LIN {X 0,Y 329.988,Z 321.354,A -85,B 0,C 180,E1 16556.004,E2 16556.004} C_VEL
LIN {X 0,Y 330.001,Z 321.346,A -85,B 0,C 180,E1 16551.813,E2 16551.813} C_VEL
LIN {X 0,Y 330.018,Z 321.353,A -85,B 0,C 180,E1 16547.578,E2 16547.578} C_VEL
LIN {X 0,Y 330.031,Z 321.366,A -85,B 0,C 180,E1 16543.273,E2 16543.273} C_VEL
LIN {X 0,Y 330.021,Z 321.374,A -85,B 0,C 180,E1 16538.867,E2 16538.867} C_VEL
LIN {X 0,Y 330.018,Z 321.377,A -85,B 0,C 180,E1 16534.711,E2 16534.711} C_VEL
LIN {X 0,Y 330.082,Z 321.657,A -85,B 0,C 180,E1 16533.325,E2 16533.325} C_VEL
LIN {X 0,Y 331.592,Z 325.229,A -85,B 0,C 180,E1 16532.136,E2 16532.136} C_VEL
LIN {X 0,Y 332.907,Z 326.905,A -85,B 0,C 180,E1 16531.475,E2 16531.475} C_VEL
LIN {X 0,Y 334.885,Z 330.792,A -85,B 0,C 180,E1 16530.29,E2 16530.29} C_VEL
LIN {X 0,Y 336.066,Z 333.043,A -85,B 0,C 180,E1 16529.617,E2 16529.617} C_VEL
LIN {X 0,Y 338.831,Z 338.21,A -85,B 0,C 180,E1 16528.116,E2 16528.116} C_VEL
LIN {X 0,Y 344.725,Z 349.404,A -85,B 0,C 180,E1 16525.153,E2 16525.153} C_VEL
LIN {X 0,Y 351.794,Z 364.539,A -85,B 0,C 180,E1 16521.714,E2 16521.714} C_VEL
LIN {X 0,Y 357.569,Z 377.862,A -85,B 0,C 180,E1 16519.132,E2 16519.132} C_VEL
LIN {X 0,Y 368.259,Z 396.802,A -85,B 0,C 180,E1 16516.934,E2 16516.934} C_VEL
LIN {X 0,Y 369.574,Z 399.796,A -85,B 0,C 180,E1 16516.66,E2 16516.66} C_VEL
LIN {X 0,Y 371.855,Z 431.34,A -85,B 0,C 180,E1 16515.478,E2 16515.478} C_VEL
LIN {X 0,Y 362.986,Z 630.851,A -85,B 0,C 180,E1 16511.25,E2 16511.25} C_VEL
LIN {X 0,Y 360.899,Z 652.81,A -85,B 0,C 180,E1 16510.527,E2 16510.527} C_VEL
LIN {X 0,Y 357.99,Z 673.843,A -85,B 0,C 180,E1 16509.552,E2 16509.552} C_VEL
LIN {X 0,Y 354.589,Z 694.236,A -85,B 0,C 180,E1 16508.28,E2 16508.28} C_VEL
LIN {X 0,Y 350.954,Z 713.405,A -85,B 0,C 180,E1 16506.746,E2 16506.746} C_VEL
LIN {X 0,Y 347.238,Z 731.415,A -85,B 0,C 180,E1 16504.959,E2 16504.959} C_VEL
LIN {X 0,Y 343.48,Z 748.656,A -85,B 0,C 180,E1 16502.88,E2 16502.88} C_VEL
LIN {X 0,Y 339.836,Z 765.3,A -85,B 0,C 180,E1 16500.452,E2 16500.452} C_VEL
LIN {X 0,Y 336.55,Z 780.44,A -85,B 0,C 180,E1 16497.802,E2 16497.802} C_VEL
LIN {X 0,Y 333.831,Z 793.946,A -85,B 0,C 180,E1 16494.98,E2 16494.98} C_VEL
LIN {X 0,Y 331.667,Z 806.101,A -85,B 0,C 180,E1 16491.95,E2 16491.95} C_VEL
LIN {X 0,Y 330.113,Z 816.843,A -85,B 0,C 180,E1 16488.726,E2 16488.726} C_VEL
LIN {X 0,Y 329.206,Z 826.04,A -85,B 0,C 180,E1 16485.321,E2 16485.321} C_VEL
LIN {X 0,Y 328.863,Z 833.265,A -85,B 0,C 180,E1 16481.931,E2 16481.931} C_VEL
LIN {X 0,Y 328.935,Z 838.668,A -85,B 0,C 180,E1 16478.565,E2 16478.565} C_VEL
LIN {X 0,Y 329.19,Z 842.319,A -85,B 0,C 180,E1 16475.228,E2 16475.228} C_VEL
LIN {X 0,Y 329.381,Z 844.1,A -85,B 0,C 180,E1 16472.262,E2 16472.262} C_VEL
LIN {X 0,Y 329.434,Z 844.424,A -85,B 0,C 180,E1 16469.13,E2 16469.13} C_VEL
LIN {X 0,Y 329.272,Z 843.237,A -85,B 0,C 180,E1 16465.995,E2 16465.995} C_VEL
LIN {X 0,Y 329.027,Z 840.42,A -85,B 0,C 180,E1 16462.843,E2 16462.843} C_VEL
LIN {X 0,Y 328.865,Z 835.744,A -85,B 0,C 180,E1 16459.49,E2 16459.49} C_VEL
LIN {X 0,Y 329.002,Z 829.277,A -85,B 0,C 180,E1 16456.109,E2 16456.109} C_VEL
LIN {X 0,Y 329.612,Z 821.315,A -85,B 0,C 180,E1 16452.848,E2 16452.848} C_VEL
LIN {X 0,Y 330.897,Z 811.117,A -85,B 0,C 180,E1 16449.482,E2 16449.482} C_VEL
LIN {X 0,Y 332.85,Z 799.201,A -85,B 0,C 180,E1 16446.264,E2 16446.264} C_VEL
LIN {X 0,Y 335.449,Z 785.75,A -85,B 0,C 180,E1 16443.252,E2 16443.252} C_VEL
LIN {X 0,Y 338.62,Z 770.765,A -85,B 0,C 180,E1 16440.456,E2 16440.456} C_VEL
LIN {X 0,Y 341.998,Z 755.34,A -85,B 0,C 180,E1 16438.052,E2 16438.052} C_VEL
LIN {X 0,Y 345.669,Z 738.547,A -85,B 0,C 180,E1 16435.866,E2 16435.866} C_VEL
LIN {X 0,Y 349.551,Z 720.157,A -85,B 0,C 180,E1 16433.898,E2 16433.898} C_VEL
LIN {X 0,Y 353.319,Z 700.736,A -85,B 0,C 180,E1 16432.218,E2 16432.218} C_VEL
LIN {X 0,Y 356.709,Z 681.467,A -85,B 0,C 180,E1 16430.901,E2 16430.901} C_VEL
LIN {X 0,Y 359.711,Z 661.609,A -85,B 0,C 180,E1 16429.858,E2 16429.858} C_VEL
LIN {X 0,Y 362.13,Z 640.669,A -85,B 0,C 180,E1 16429.053,E2 16429.053} C_VEL
LIN {X 0,Y 363.596,Z 618.696,A -85,B 0,C 180,E1 16428.472,E2 16428.472} C_VEL
LIN {X 0,Y 371.808,Z 429.248,A -85,B 0,C 180,E1 16424.483,E2 16424.483} C_VEL
LIN {X 0,Y 369.242,Z 398.809,A -85,B 0,C 180,E1 16423.296,E2 16423.296} C_VEL
LIN {X 0,Y 359.659,Z 381.559,A -85,B 0,C 180,E1 16421.345,E2 16421.345} C_VEL
LIN {X 0,Y 357.005,Z 376.819,A -85,B 0,C 180,E1 16420.734,E2 16420.734} C_VEL
LIN {X 0,Y 350.035,Z 360.556,A -85,B 0,C 180,E1 16417.432,E2 16417.432} C_VEL
LIN {X 0,Y 343.951,Z 348.039,A -85,B 0,C 180,E1 16414.531,E2 16414.531} C_VEL
LIN {X 0,Y 339.399,Z 339.27,A -85,B 0,C 180,E1 16412.223,E2 16412.223} C_VEL
LIN {X 0,Y 337.08,Z 334.954,A -85,B 0,C 180,E1 16410.994,E2 16410.994} C_VEL
LIN {X 0,Y 335.156,Z 331.101,A -85,B 0,C 180,E1 16409.881,E2 16409.881} C_VEL
LIN {X 0,Y 333.053,Z 327.414,A -85,B 0,C 180,E1 16408.707,E2 16408.707} C_VEL
LIN {X 0,Y 332.535,Z 326.256,A -85,B 0,C 180,E1 16408.364,E2 16408.364} C_VEL
LIN {X 0,Y 330.422,Z 323.03,A -85,B 0,C 180,E1 16407.189,E2 16407.189} C_VEL
LIN {X 0,Y 330.046,Z 321.433,A -85,B 0,C 180,E1 16406.581,E2 16406.581} C_VEL
LIN {X 0,Y 330.017,Z 321.356,A -85,B 0,C 180,E1 16402.254,E2 16402.254} C_VEL
LIN {X 0,Y 330.003,Z 321.353,A -85,B 0,C 180,E1 16397.947,E2 16397.947} C_VEL
LIN {X 0,Y 329.993,Z 321.349,A -85,B 0,C 180,E1 16393.67,E2 16393.67} C_VEL
LIN {X 0,Y 329.991,Z 321.356,A -85,B 0,C 180,E1 16389.417,E2 16389.417} C_VEL
LIN {X 0,Y 329.993,Z 321.38,A -85,B 0,C 180,E1 16385.215,E2 16385.215} C_VEL
LIN {X 0,Y 330.002,Z 321.367,A -85,B 0,C 180,E1 16380.868,E2 16380.868} C_VEL
LIN {X 0,Y 330.005,Z 321.345,A -85,B 0,C 180,E1 16376.504,E2 16376.504} C_VEL
LIN {X 0,Y 330.01,Z 321.346,A -85,B 0,C 180,E1 16372.163,E2 16372.163} C_VEL
LIN {X 0,Y 330.002,Z 321.376,A -85,B 0,C 180,E1 16367.932,E2 16367.932} C_VEL
LIN {X 0,Y 329.999,Z 321.371,A -85,B 0,C 180,E1 16363.633,E2 16363.633} C_VEL
LIN {X 0,Y 329.996,Z 321.355,A -85,B 0,C 180,E1 16359.237,E2 16359.237} C_VEL
LIN {X 0,Y 330.003,Z 321.349,A -85,B 0,C 180,E1 16354.901,E2 16354.901} C_VEL
LIN {X 0,Y 330.014,Z 321.352,A -85,B 0,C 180,E1 16350.755,E2 16350.755} C_VEL
LIN {X 0,Y 330.024,Z 321.355,A -85,B 0,C 180,E1 16346.537,E2 16346.537} C_VEL
LIN {X 0,Y 330.063,Z 321.623,A -85,B 0,C 180,E1 16344.507,E2 16344.507} C_VEL
LIN {X 0,Y 331.69,Z 325.358,A -85,B 0,C 180,E1 16343.139,E2 16343.139} C_VEL
LIN {X 0,Y 332.674,Z 327.051,A -85,B 0,C 180,E1 16342.508,E2 16342.508} C_VEL
LIN {X 0,Y 335.181,Z 332.261,A -85,B 0,C 180,E1 16340.772,E2 16340.772} C_VEL
LIN {X 0,Y 338.644,Z 339.138,A -85,B 0,C 180,E1 16338.584,E2 16338.584} C_VEL
LIN {X 0,Y 343.572,Z 350.049,A -85,B 0,C 180,E1 16335.581,E2 16335.581} C_VEL
LIN {X 0,Y 354.646,Z 366.45,A -85,B 0,C 180,E1 16333.096,E2 16333.096} C_VEL
LIN {X 0,Y 365.235,Z 383.822,A -85,B 0,C 180,E1 16330.924,E2 16330.924} C_VEL
LIN {X 0,Y 371.372,Z 395.131,A -85,B 0,C 180,E1 16329.731,E2 16329.731} C_VEL
LIN {X 0,Y 365.497,Z 566.215,A -85,B 0,C 180,E1 16326.469,E2 16326.469} C_VEL
LIN {X 0,Y 364.483,Z 584.95,A -85,B 0,C 180,E1 16325.856,E2 16325.856} C_VEL
LIN {X 0,Y 362.848,Z 602.649,A -85,B 0,C 180,E1 16325.023,E2 16325.023} C_VEL
LIN {X 0,Y 360.528,Z 620.805,A -85,B 0,C 180,E1 16323.878,E2 16323.878} C_VEL
LIN {X 0,Y 357.652,Z 638.242,A -85,B 0,C 180,E1 16322.462,E2 16322.462} C_VEL
LIN {X 0,Y 354.406,Z 654.561,A -85,B 0,C 180,E1 16320.8,E2 16320.8} C_VEL
LIN {X 0,Y 350.903,Z 669.814,A -85,B 0,C 180,E1 16318.879,E2 16318.879} C_VEL
LIN {X 0,Y 347.276,Z 683.981,A -85,B 0,C 180,E1 16316.688,E2 16316.688} C_VEL
LIN {X 0,Y 343.882,Z 696.2,A -85,B 0,C 180,E1 16314.385,E2 16314.385} C_VEL
LIN {X 0,Y 340.482,Z 707.778,A -85,B 0,C 180,E1 16311.716,E2 16311.716} C_VEL
LIN {X 0,Y 337.476,Z 717.82,A -85,B 0,C 180,E1 16308.84,E2 16308.84} C_VEL
LIN {X 0,Y 334.91,Z 726.341,A -85,B 0,C 180,E1 16305.764,E2 16305.764} C_VEL
LIN {X 0,Y 332.895,Z 733.313,A -85,B 0,C 180,E1 16302.489,E2 16302.489} C_VEL
LIN {X 0,Y 331.513,Z 738.445,A -85,B 0,C 180,E1 16299.198,E2 16299.198} C_VEL
LIN {X 0,Y 330.607,Z 742.054,A -85,B 0,C 180,E1 16295.728,E2 16295.728} C_VEL
LIN {X 0,Y 330.182,Z 743.952,A -85,B 0,C 180,E1 16292.256,E2 16292.256} C_VEL
LIN {X 0,Y 330.123,Z 744.22,A -85,B 0,C 180,E1 16288.785,E2 16288.785} C_VEL
LIN {X 0,Y 330.425,Z 742.87,A -85,B 0,C 180,E1 16285.314,E2 16285.314} C_VEL
LIN {X 0,Y 331.162,Z 739.844,A -85,B 0,C 180,E1 16281.842,E2 16281.842} C_VEL
LIN {X 0,Y 332.361,Z 735.3,A -85,B 0,C 180,E1 16278.548,E2 16278.548} C_VEL
LIN {X 0,Y 334.15,Z 728.997,A -85,B 0,C 180,E1 16275.266,E2 16275.266} C_VEL
LIN {X 0,Y 336.491,Z 721.192,A -85,B 0,C 180,E1 16272.179,E2 16272.179} C_VEL
LIN {X 0,Y 337.17,Z 718.967,A -85,B 0,C 180,E1 16271.419,E2 16271.419} C_VEL
LIN {X 0,Y 337.295,Z 715.6,A -85,B 0,C 180,E1 16270.238,E2 16270.238} C_VEL
LIN {X 0,Y 334.749,Z 706.748,A -85,B 0,C 180,E1 16267.184,E2 16267.184} C_VEL
LIN {X 0,Y 335.198,Z 702.513,A -85,B 0,C 180,E1 16266.068,E2 16266.068} C_VEL
LIN {X 0,Y 338.821,Z 690.407,A -85,B 0,C 180,E1 16263.539,E2 16263.539} C_VEL
LIN {X 0,Y 342.603,Z 676.785,A -85,B 0,C 180,E1 16261.215,E2 16261.215} C_VEL
LIN {X 0,Y 346.299,Z 662.101,A -85,B 0,C 180,E1 16259.171,E2 16259.171} C_VEL
LIN {X 0,Y 349.849,Z 646.05,A -85,B 0,C 180,E1 16257.358,E2 16257.358} C_VEL
LIN {X 0,Y 352.911,Z 629.764,A -85,B 0,C 180,E1 16255.878,E2 16255.878} C_VEL
LIN {X 0,Y 355.587,Z 612.062,A -85,B 0,C 180,E1 16254.604,E2 16254.604} C_VEL
LIN {X 0,Y 357.708,Z 593.156,A -85,B 0,C 180,E1 16253.573,E2 16253.573} C_VEL
LIN {X 0,Y 359.098,Z 573.733,A -85,B 0,C 180,E1 16252.823,E2 16252.823} C_VEL
LIN {X 0,Y 359.921,Z 549.235,A -85,B 0,C 180,E1 16252.243,E2 16252.243} C_VEL
LIN {X 0,Y 365.403,Z 397.808,A -85,B 0,C 180,E1 16249.34,E2 16249.34} C_VEL
LIN {X 0,Y 355.071,Z 379.673,A -85,B 0,C 180,E1 16247.215,E2 16247.215} C_VEL
LIN {X 0,Y 345.298,Z 364.445,A -85,B 0,C 180,E1 16245.06,E2 16245.06} C_VEL
LIN {X 0,Y 335.772,Z 350.784,A -85,B 0,C 180,E1 16242.761,E2 16242.761} C_VEL
LIN {X 0,Y 331.864,Z 342.522,A -85,B 0,C 180,E1 16240.339,E2 16240.339} C_VEL
LIN {X 0,Y 328.69,Z 335.771,A -85,B 0,C 180,E1 16238.135,E2 16238.135} C_VEL
LIN {X 0,Y 326.623,Z 331.539,A -85,B 0,C 180,E1 16236.651,E2 16236.651} C_VEL
LIN {X 0,Y 324.81,Z 328.032,A -85,B 0,C 180,E1 16235.341,E2 16235.341} C_VEL
LIN {X 0,Y 322.269,Z 323.301,A -85,B 0,C 180,E1 16233.43,E2 16233.43} C_VEL
LIN {X 0,Y 322.076,Z 322.376,A -85,B 0,C 180,E1 16232.907,E2 16232.907} C_VEL
LIN {X 0,Y 322.074,Z 322.345,A -85,B 0,C 180,E1 16228.535,E2 16228.535} C_VEL
LIN {X 0,Y 322.084,Z 322.337,A -85,B 0,C 180,E1 16224.126,E2 16224.126} C_VEL
LIN {X 0,Y 322.092,Z 322.332,A -85,B 0,C 180,E1 16219.778,E2 16219.778} C_VEL
LIN {X 0,Y 322.088,Z 322.339,A -85,B 0,C 180,E1 16215.484,E2 16215.484} C_VEL
LIN {X 0,Y 322.064,Z 322.365,A -85,B 0,C 180,E1 16211.098,E2 16211.098} C_VEL
LIN {X 0,Y 322.048,Z 322.354,A -85,B 0,C 180,E1 16206.776,E2 16206.776} C_VEL
LIN {X 0,Y 322.04,Z 322.336,A -85,B 0,C 180,E1 16202.314,E2 16202.314} C_VEL
LIN {X 0,Y 322.046,Z 322.337,A -85,B 0,C 180,E1 16198.043,E2 16198.043} C_VEL
LIN {X 0,Y 322.081,Z 322.351,A -85,B 0,C 180,E1 16193.584,E2 16193.584} C_VEL
LIN {X 0,Y 322.082,Z 322.365,A -85,B 0,C 180,E1 16189.266,E2 16189.266} C_VEL
LIN {X 0,Y 322.069,Z 322.351,A -85,B 0,C 180,E1 16184.884,E2 16184.884} C_VEL
LIN {X 0,Y 322.064,Z 322.345,A -85,B 0,C 180,E1 16180.599,E2 16180.599} C_VEL
LIN {X 0,Y 322.066,Z 322.345,A -85,B 0,C 180,E1 16176.198,E2 16176.198} C_VEL
LIN {X 0,Y 322.141,Z 322.707,A -85,B 0,C 180,E1 16175.522,E2 16175.522} C_VEL
LIN {X 0,Y 323.78,Z 326.39,A -85,B 0,C 180,E1 16174.188,E2 16174.188} C_VEL
LIN {X 0,Y 325.054,Z 327.877,A -85,B 0,C 180,E1 16173.512,E2 16173.512} C_VEL
LIN {X 0,Y 326.832,Z 331.6,A -85,B 0,C 180,E1 16172.29,E2 16172.29} C_VEL
LIN {X 0,Y 328.017,Z 333.531,A -85,B 0,C 180,E1 16171.607,E2 16171.607} C_VEL
LIN {X 0,Y 330.931,Z 338.973,A -85,B 0,C 180,E1 16169.898,E2 16169.898} C_VEL
LIN {X 0,Y 335.271,Z 347.087,A -85,B 0,C 180,E1 16167.534,E2 16167.534} C_VEL
LIN {X 0,Y 341.078,Z 358.854,A -85,B 0,C 180,E1 16164.52,E2 16164.52} C_VEL
LIN {X 0,Y 347.447,Z 373.012,A -85,B 0,C 180,E1 16161.357,E2 16161.357} C_VEL
LIN {X 0,Y 349.493,Z 377.491,A -85,B 0,C 180,E1 16160.519,E2 16160.519} C_VEL
LIN {X 0,Y 359.941,Z 395.515,A -85,B 0,C 180,E1 16158.242,E2 16158.242} C_VEL
LIN {X 0,Y 363.916,Z 403.32,A -85,B 0,C 180,E1 16157.407,E2 16157.407} C_VEL
LIN {X 0,Y 365.906,Z 432.308,A -85,B 0,C 180,E1 16156.299,E2 16156.299} C_VEL
LIN {X 0,Y 356.749,Z 630.067,A -85,B 0,C 180,E1 16152.06,E2 16152.06} C_VEL
LIN {X 0,Y 354.599,Z 651.964,A -85,B 0,C 180,E1 16151.331,E2 16151.331} C_VEL
LIN {X 0,Y 351.557,Z 673.11,A -85,B 0,C 180,E1 16150.341,E2 16150.341} C_VEL
LIN {X 0,Y 348.102,Z 693.035,A -85,B 0,C 180,E1 16149.084,E2 16149.084} C_VEL
LIN {X 0,Y 344.385,Z 711.851,A -85,B 0,C 180,E1 16147.566,E2 16147.566} C_VEL
LIN {X 0,Y 340.48,Z 729.939,A -85,B 0,C 180,E1 16145.758,E2 16145.758} C_VEL
LIN {X 0,Y 336.537,Z 747.239,A -85,B 0,C 180,E1 16143.647,E2 16143.647} C_VEL
LIN {X 0,Y 332.731,Z 763.666,A -85,B 0,C 180,E1 16141.221,E2 16141.221} C_VEL
LIN {X 0,Y 329.186,Z 779.091,A -85,B 0,C 180,E1 16138.48,E2 16138.48} C_VEL
LIN {X 0,Y 326.291,Z 792.623,A -85,B 0,C 180,E1 16135.598,E2 16135.598} C_VEL
LIN {X 0,Y 323.958,Z 804.798,A -85,B 0,C 180,E1 16132.501,E2 16132.501} C_VEL
LIN {X 0,Y 322.282,Z 815.558,A -85,B 0,C 180,E1 16129.199,E2 16129.199} C_VEL
LIN {X 0,Y 321.288,Z 824.772,A -85,B 0,C 180,E1 16125.708,E2 16125.708} C_VEL
LIN {X 0,Y 320.898,Z 832.016,A -85,B 0,C 180,E1 16122.232,E2 16122.232} C_VEL
LIN {X 0,Y 320.976,Z 837.44,A -85,B 0,C 180,E1 16118.78,E2 16118.78} C_VEL
LIN {X 0,Y 321.244,Z 841.106,A -85,B 0,C 180,E1 16115.358,E2 16115.358} C_VEL
LIN {X 0,Y 321.466,Z 842.897,A -85,B 0,C 180,E1 16112.317,E2 16112.317} C_VEL
LIN {X 0,Y 321.525,Z 843.248,A -85,B 0,C 180,E1 16109.287,E2 16109.287} C_VEL
LIN {X 0,Y 321.372,Z 842.247,A -85,B 0,C 180,E1 16106.254,E2 16106.254} C_VEL
LIN {X 0,Y 321.104,Z 839.572,A -85,B 0,C 180,E1 16103.025,E2 16103.025} C_VEL
LIN {X 0,Y 320.905,Z 835.086,A -85,B 0,C 180,E1 16099.589,E2 16099.589} C_VEL
LIN {X 0,Y 320.995,Z 829.211,A -85,B 0,C 180,E1 16096.307,E2 16096.307} C_VEL
LIN {X 0,Y 321.615,Z 821.111,A -85,B 0,C 180,E1 16092.822,E2 16092.822} C_VEL
LIN {X 0,Y 322.849,Z 811.545,A -85,B 0,C 180,E1 16089.516,E2 16089.516} C_VEL
LIN {X 0,Y 324.686,Z 800.665,A -85,B 0,C 180,E1 16086.402,E2 16086.402} C_VEL
LIN {X 0,Y 327.285,Z 787.743,A -85,B 0,C 180,E1 16083.316,E2 16083.316} C_VEL
LIN {X 0,Y 330.473,Z 773.361,A -85,B 0,C 180,E1 16080.452,E2 16080.452} C_VEL
LIN {X 0,Y 334.021,Z 758.021,A -85,B 0,C 180,E1 16077.901,E2 16077.901} C_VEL
LIN {X 0,Y 337.894,Z 741.294,A -85,B 0,C 180,E1 16075.586,E2 16075.586} C_VEL
LIN {X 0,Y 341.994,Z 723.02,A -85,B 0,C 180,E1 16073.513,E2 16073.513} C_VEL
LIN {X 0,Y 345.892,Z 704.249,A -85,B 0,C 180,E1 16071.787,E2 16071.787} C_VEL
LIN {X 0,Y 349.539,Z 684.748,A -85,B 0,C 180,E1 16070.367,E2 16070.367} C_VEL
LIN {X 0,Y 352.746,Z 665.005,A -85,B 0,C 180,E1 16069.26,E2 16069.26} C_VEL
LIN {X 0,Y 355.371,Z 644.534,A -85,B 0,C 180,E1 16068.409,E2 16068.409} C_VEL
LIN {X 0,Y 357.081,Z 623.395,A -85,B 0,C 180,E1 16067.788,E2 16067.788} C_VEL
LIN {X 0,Y 365.862,Z 430.431,A -85,B 0,C 180,E1 16063.668,E2 16063.668} C_VEL
LIN {X 0,Y 363.563,Z 402.371,A -85,B 0,C 180,E1 16062.547,E2 16062.547} C_VEL
LIN {X 0,Y 353.314,Z 383.877,A -85,B 0,C 180,E1 16060.368,E2 16060.368} C_VEL
LIN {X 0,Y 348.685,Z 375.951,A -85,B 0,C 180,E1 16059.267,E2 16059.267} C_VEL
LIN {X 0,Y 342.375,Z 361.611,A -85,B 0,C 180,E1 16056.15,E2 16056.15} C_VEL
LIN {X 0,Y 336.776,Z 350.046,A -85,B 0,C 180,E1 16053.315,E2 16053.315} C_VEL
LIN {X 0,Y 332.063,Z 341.072,A -85,B 0,C 180,E1 16050.789,E2 16050.789} C_VEL
LIN {X 0,Y 329.674,Z 336.622,A -85,B 0,C 180,E1 16049.427,E2 16049.427} C_VEL
LIN {X 0,Y 327.403,Z 332.26,A -85,B 0,C 180,E1 16048.048,E2 16048.048} C_VEL
LIN {X 0,Y 325.38,Z 328.95,A -85,B 0,C 180,E1 16046.853,E2 16046.853} C_VEL
LIN {X 0,Y 324.665,Z 327.308,A -85,B 0,C 180,E1 16046.325,E2 16046.325} C_VEL
LIN {X 0,Y 322.623,Z 324.406,A -85,B 0,C 180,E1 16045.124,E2 16045.124} C_VEL
LIN {X 0,Y 322.127,Z 322.599,A -85,B 0,C 180,E1 16044.48,E2 16044.48} C_VEL
LIN {X 0,Y 322.095,Z 322.363,A -85,B 0,C 180,E1 16040.535,E2 16040.535} C_VEL
LIN {X 0,Y 322.076,Z 322.366,A -85,B 0,C 180,E1 16036.224,E2 16036.224} C_VEL
LIN {X 0,Y 322.06,Z 322.349,A -85,B 0,C 180,E1 16032.005,E2 16032.005} C_VEL
LIN {X 0,Y 322.048,Z 322.338,A -85,B 0,C 180,E1 16027.672,E2 16027.672} C_VEL
LIN {X 0,Y 322.043,Z 322.338,A -85,B 0,C 180,E1 16023.381,E2 16023.381} C_VEL
LIN {X 0,Y 322.048,Z 322.359,A -85,B 0,C 180,E1 16019.11,E2 16019.11} C_VEL
LIN {X 0,Y 322.069,Z 322.364,A -85,B 0,C 180,E1 16014.656,E2 16014.656} C_VEL
LIN {X 0,Y 322.075,Z 322.336,A -85,B 0,C 180,E1 16010.349,E2 16010.349} C_VEL
LIN {X 0,Y 322.068,Z 322.333,A -85,B 0,C 180,E1 16005.986,E2 16005.986} C_VEL
LIN {X 0,Y 322.066,Z 322.347,A -85,B 0,C 180,E1 16001.726,E2 16001.726} C_VEL
LIN {X 0,Y 322.061,Z 322.365,A -85,B 0,C 180,E1 15997.358,E2 15997.358} C_VEL
LIN {X 0,Y 322.072,Z 322.368,A -85,B 0,C 180,E1 15992.847,E2 15992.847} C_VEL
LIN {X 0,Y 322.087,Z 322.36,A -85,B 0,C 180,E1 15988.565,E2 15988.565} C_VEL
LIN {X 0,Y 322.124,Z 322.658,A -85,B 0,C 180,E1 15986.674,E2 15986.674} C_VEL
LIN {X 0,Y 323.828,Z 326.438,A -85,B 0,C 180,E1 15985.165,E2 15985.165} C_VEL
LIN {X 0,Y 324.865,Z 328.259,A -85,B 0,C 180,E1 15984.429,E2 15984.429} C_VEL
LIN {X 0,Y 327.192,Z 332.729,A -85,B 0,C 180,E1 15982.766,E2 15982.766} C_VEL
LIN {X 0,Y 331.233,Z 340.957,A -85,B 0,C 180,E1 15979.987,E2 15979.987} C_VEL
LIN {X 0,Y 335.521,Z 350.368,A -85,B 0,C 180,E1 15977.199,E2 15977.199} C_VEL
LIN {X 0,Y 344.557,Z 363.411,A -85,B 0,C 180,E1 15974.981,E2 15974.981} C_VEL
LIN {X 0,Y 353.664,Z 377.534,A -85,B 0,C 180,E1 15972.956,E2 15972.956} C_VEL
LIN {X 0,Y 364.235,Z 395.671,A -85,B 0,C 180,E1 15970.776,E2 15970.776} C_VEL
LIN {X 0,Y 365.435,Z 398.292,A -85,B 0,C 180,E1 15970.528,E2 15970.528} C_VEL
LIN {X 0,Y 359.336,Z 566.906,A -85,B 0,C 180,E1 15967.269,E2 15967.269} C_VEL
LIN {X 0,Y 358.271,Z 585.725,A -85,B 0,C 180,E1 15966.646,E2 15966.646} C_VEL
LIN {X 0,Y 356.526,Z 603.807,A -85,B 0,C 180,E1 15965.782,E2 15965.782} C_VEL
LIN {X 0,Y 354.199,Z 621.302,A -85,B 0,C 180,E1 15964.666,E2 15964.666} C_VEL
LIN {X 0,Y 351.205,Z 638.841,A -85,B 0,C 180,E1 15963.231,E2 15963.231} C_VEL
LIN {X 0,Y 347.815,Z 655.243,A -85,B 0,C 180,E1 15961.546,E2 15961.546} C_VEL
LIN {X 0,Y 344.163,Z 670.564,A -85,B 0,C 180,E1 15959.595,E2 15959.595} C_VEL
LIN {X 0,Y 340.5,Z 684.31,A -85,B 0,C 180,E1 15957.452,E2 15957.452} C_VEL
LIN {X 0,Y 336.691,Z 697.465,A -85,B 0,C 180,E1 15954.941,E2 15954.941} C_VEL
LIN {X 0,Y 333.135,Z 709.024,A -85,B 0,C 180,E1 15952.22,E2 15952.22} C_VEL
LIN {X 0,Y 329.981,Z 719.051,A -85,B 0,C 180,E1 15949.285,E2 15949.285} C_VEL
LIN {X 0,Y 327.283,Z 727.563,A -85,B 0,C 180,E1 15946.141,E2 15946.141} C_VEL
LIN {X 0,Y 325.156,Z 734.527,A -85,B 0,C 180,E1 15942.791,E2 15942.791} C_VEL
LIN {X 0,Y 323.692,Z 739.654,A -85,B 0,C 180,E1 15939.422,E2 15939.422} C_VEL
LIN {X 0,Y 322.732,Z 743.258,A -85,B 0,C 180,E1 15935.868,E2 15935.868} C_VEL
LIN {X 0,Y 322.279,Z 745.154,A -85,B 0,C 180,E1 15932.311,E2 15932.311} C_VEL
LIN {X 0,Y 322.215,Z 745.422,A -85,B 0,C 180,E1 15928.755,E2 15928.755} C_VEL
LIN {X 0,Y 322.536,Z 744.073,A -85,B 0,C 180,E1 15925.199,E2 15925.199} C_VEL
LIN {X 0,Y 323.32,Z 741.048,A -85,B 0,C 180,E1 15921.643,E2 15921.643} C_VEL
LIN {X 0,Y 324.591,Z 736.51,A -85,B 0,C 180,E1 15918.27,E2 15918.27} C_VEL
LIN {X 0,Y 326.483,Z 730.211,A -85,B 0,C 180,E1 15914.912,E2 15914.912} C_VEL
LIN {X 0,Y 328.949,Z 722.415,A -85,B 0,C 180,E1 15911.756,E2 15911.756} C_VEL
LIN {X 0,Y 331.87,Z 713.174,A -85,B 0,C 180,E1 15908.806,E2 15908.806} C_VEL
LIN {X 0,Y 335.198,Z 702.513,A -85,B 0,C 180,E1 15906.068,E2 15906.068} C_VEL
LIN {X 0,Y 335.725,Z 698.146,A -85,B 0,C 180,E1 15904.973,E2 15904.973} C_VEL
LIN {X 0,Y 334.106,Z 687.632,A -85,B 0,C 180,E1 15902.275,E2 15902.275} C_VEL
LIN {X 0,Y 334.506,Z 682.533,A -85,B 0,C 180,E1 15901.275,E2 15901.275} C_VEL
LIN {X 0,Y 334.7,Z 681.744,A -85,B 0,C 180,E1 15901.146,E2 15901.146} C_VEL
LIN {X 0,Y 338.614,Z 667.296,A -85,B 0,C 180,E1 15898.986,E2 15898.986} C_VEL
LIN {X 0,Y 342.34,Z 651.752,A -85,B 0,C 180,E1 15897.096,E2 15897.096} C_VEL
LIN {X 0,Y 345.87,Z 634.511,A -85,B 0,C 180,E1 15895.417,E2 15895.417} C_VEL
LIN {X 0,Y 348.705,Z 617.506,A -85,B 0,C 180,E1 15894.101,E2 15894.101} C_VEL
LIN {X 0,Y 351.098,Z 598.691,A -85,B 0,C 180,E1 15892.985,E2 15892.985} C_VEL
LIN {X 0,Y 352.734,Z 579.403,A -85,B 0,C 180,E1 15892.157,E2 15892.157} C_VEL
LIN {X 0,Y 353.592,Z 559.428,A -85,B 0,C 180,E1 15891.603,E2 15891.603} C_VEL
LIN {X 0,Y 359.51,Z 400.832,A -85,B 0,C 180,E1 15888.507,E2 15888.507} C_VEL
LIN {X 0,Y 349.361,Z 383.174,A -85,B 0,C 180,E1 15886.333,E2 15886.333} C_VEL
LIN {X 0,Y 340.387,Z 369.124,A -85,B 0,C 180,E1 15884.268,E2 15884.268} C_VEL
LIN {X 0,Y 331.339,Z 356.057,A -85,B 0,C 180,E1 15882.003,E2 15882.003} C_VEL
LIN {X 0,Y 327.737,Z 351.036,A -85,B 0,C 180,E1 15880.99,E2 15880.99} C_VEL
LIN {X 0,Y 323.667,Z 342.153,A -85,B 0,C 180,E1 15878.159,E2 15878.159} C_VEL
LIN {X 0,Y 320.744,Z 336.628,A -85,B 0,C 180,E1 15876.099,E2 15876.099} C_VEL
LIN {X 0,Y 318.81,Z 332.641,A -85,B 0,C 180,E1 15874.587,E2 15874.587} C_VEL
LIN {X 0,Y 316.469,Z 328.067,A -85,B 0,C 180,E1 15872.702,E2 15872.702} C_VEL
LIN {X 0,Y 314.358,Z 324.467,A -85,B 0,C 180,E1 15871.016,E2 15871.016} C_VEL
LIN {X 0,Y 314.145,Z 323.364,A -85,B 0,C 180,E1 15870.4,E2 15870.4} C_VEL
LIN {X 0,Y 314.152,Z 323.333,A -85,B 0,C 180,E1 15866.054,E2 15866.054} C_VEL
LIN {X 0,Y 314.166,Z 323.343,A -85,B 0,C 180,E1 15861.665,E2 15861.665} C_VEL
LIN {X 0,Y 314.136,Z 323.353,A -85,B 0,C 180,E1 15857.218,E2 15857.218} C_VEL
LIN {X 0,Y 314.117,Z 323.332,A -85,B 0,C 180,E1 15852.875,E2 15852.875} C_VEL
LIN {X 0,Y 314.108,Z 323.321,A -85,B 0,C 180,E1 15848.42,E2 15848.42} C_VEL
LIN {X 0,Y 314.115,Z 323.328,A -85,B 0,C 180,E1 15844.016,E2 15844.016} C_VEL
LIN {X 0,Y 314.135,Z 323.35,A -85,B 0,C 180,E1 15839.636,E2 15839.636} C_VEL
LIN {X 0,Y 314.13,Z 323.341,A -85,B 0,C 180,E1 15835.253,E2 15835.253} C_VEL
LIN {X 0,Y 314.119,Z 323.327,A -85,B 0,C 180,E1 15830.843,E2 15830.843} C_VEL
LIN {X 0,Y 314.115,Z 323.325,A -85,B 0,C 180,E1 15826.376,E2 15826.376} C_VEL
LIN {X 0,Y 314.123,Z 323.329,A -85,B 0,C 180,E1 15822.016,E2 15822.016} C_VEL
LIN {X 0,Y 314.163,Z 323.599,A -85,B 0,C 180,E1 15818.139,E2 15818.139} C_VEL
LIN {X 0,Y 315.937,Z 327.481,A -85,B 0,C 180,E1 15816.5,E2 15816.5} C_VEL
LIN {X 0,Y 317.329,Z 329.355,A -85,B 0,C 180,E1 15815.622,E2 15815.622} C_VEL
LIN {X 0,Y 319.354,Z 333.115,A -85,B 0,C 180,E1 15814.203,E2 15814.203} C_VEL
LIN {X 0,Y 320.252,Z 334.58,A -85,B 0,C 180,E1 15813.639,E2 15813.639} C_VEL
LIN {X 0,Y 322.938,Z 339.463,A -85,B 0,C 180,E1 15811.926,E2 15811.926} C_VEL
LIN {X 0,Y 327.639,Z 348.178,A -85,B 0,C 180,E1 15809.157,E2 15809.157} C_VEL
LIN {X 0,Y 333.815,Z 360.651,A -85,B 0,C 180,E1 15805.729,E2 15805.729} C_VEL
LIN {X 0,Y 340.38,Z 375.126,A -85,B 0,C 180,E1 15802.339,E2 15802.339} C_VEL
LIN {X 0,Y 349.582,Z 390.621,A -85,B 0,C 180,E1 15800.105,E2 15800.105} C_VEL
LIN {X 0,Y 358.311,Z 406.665,A -85,B 0,C 180,E1 15798.184,E2 15798.184} C_VEL
LIN {X 0,Y 360.026,Z 433.456,A -85,B 0,C 180,E1 15797.144,E2 15797.144} C_VEL
LIN {X 0,Y 350.599,Z 629.113,A -85,B 0,C 180,E1 15792.904,E2 15792.904} C_VEL
LIN {X 0,Y 348.388,Z 650.993,A -85,B 0,C 180,E1 15792.168,E2 15792.168} C_VEL
LIN {X 0,Y 345.208,Z 672.311,A -85,B 0,C 180,E1 15791.162,E2 15791.162} C_VEL
LIN {X 0,Y 341.563,Z 692.518,A -85,B 0,C 180,E1 15789.871,E2 15789.871} C_VEL
LIN {X 0,Y 337.601,Z 711.697,A -85,B 0,C 180,E1 15788.295,E2 15788.295} C_VEL
LIN {X 0,Y 333.449,Z 730.002,A -85,B 0,C 180,E1 15786.419,E2 15786.419} C_VEL
LIN {X 0,Y 329.348,Z 747.107,A -85,B 0,C 180,E1 15784.273,E2 15784.273} C_VEL
LIN {X 0,Y 325.365,Z 763.368,A -85,B 0,C 180,E1 15781.804,E2 15781.804} C_VEL
LIN {X 0,Y 321.656,Z 778.655,A -85,B 0,C 180,E1 15779.006,E2 15779.006} C_VEL
LIN {X 0,Y 318.447,Z 792.826,A -85,B 0,C 180,E1 15775.876,E2 15775.876} C_VEL
LIN {X 0,Y 315.919,Z 805.393,A -85,B 0,C 180,E1 15772.516,E2 15772.516} C_VEL
LIN {X 0,Y 314.217,Z 815.959,A -85,B 0,C 180,E1 15769.079,E2 15769.079} C_VEL
LIN {X 0,Y 313.267,Z 824.77,A -85,B 0,C 180,E1 15765.551,E2 15765.551} C_VEL
LIN {X 0,Y 312.918,Z 831.796,A -85,B 0,C 180,E1 15761.987,E2 15761.987} C_VEL
LIN {X 0,Y 313.033,Z 836.689,A -85,B 0,C 180,E1 15758.634,E2 15758.634} C_VEL
LIN {X 0,Y 313.346,Z 840.164,A -85,B 0,C 180,E1 15755.126,E2 15755.126} C_VEL
LIN {X 0,Y 313.56,Z 841.841,A -85,B 0,C 180,E1 15752.01,E2 15752.01} C_VEL
LIN {X 0,Y 313.609,Z 841.993,A -85,B 0,C 180,E1 15748.904,E2 15748.904} C_VEL
LIN {X 0,Y 313.402,Z 840.687,A -85,B 0,C 180,E1 15745.609,E2 15745.609} C_VEL
LIN {X 0,Y 313.116,Z 837.976,A -85,B 0,C 180,E1 15742.477,E2 15742.477} C_VEL
LIN {X 0,Y 312.929,Z 833.554,A -85,B 0,C 180,E1 15739.134,E2 15739.134} C_VEL
LIN {X 0,Y 313.098,Z 827.154,A -85,B 0,C 180,E1 15735.577,E2 15735.577} C_VEL
LIN {X 0,Y 313.791,Z 819.369,A -85,B 0,C 180,E1 15732.189,E2 15732.189} C_VEL
LIN {X 0,Y 315.279,Z 809.11,A -85,B 0,C 180,E1 15728.611,E2 15728.611} C_VEL
LIN {X 0,Y 317.501,Z 797.265,A -85,B 0,C 180,E1 15725.24,E2 15725.24} C_VEL
LIN {X 0,Y 320.421,Z 783.905,A -85,B 0,C 180,E1 15722.092,E2 15722.092} C_VEL
LIN {X 0,Y 323.84,Z 769.519,A -85,B 0,C 180,E1 15719.272,E2 15719.272} C_VEL
LIN {X 0,Y 327.687,Z 753.709,A -85,B 0,C 180,E1 15716.687,E2 15716.687} C_VEL
LIN {X 0,Y 331.911,Z 736.35,A -85,B 0,C 180,E1 15714.346,E2 15714.346} C_VEL
LIN {X 0,Y 336.156,Z 717.963,A -85,B 0,C 180,E1 15712.322,E2 15712.322} C_VEL
LIN {X 0,Y 340.279,Z 698.531,A -85,B 0,C 180,E1 15710.604,E2 15710.604} C_VEL
LIN {X 0,Y 343.957,Z 679.227,A -85,B 0,C 180,E1 15709.263,E2 15709.263} C_VEL
LIN {X 0,Y 347.131,Z 659.587,A -85,B 0,C 180,E1 15708.215,E2 15708.215} C_VEL
LIN {X 0,Y 349.692,Z 638.776,A -85,B 0,C 180,E1 15707.402,E2 15707.402} C_VEL
LIN {X 0,Y 351.251,Z 616.882,A -85,B 0,C 180,E1 15706.811,E2 15706.811} C_VEL
LIN {X 0,Y 359.978,Z 431.367,A -85,B 0,C 180,E1 15702.816,E2 15702.816} C_VEL
LIN {X 0,Y 357.988,Z 406.017,A -85,B 0,C 180,E1 15701.783,E2 15701.783} C_VEL
LIN {X 0,Y 347.786,Z 387.628,A -85,B 0,C 180,E1 15699.526,E2 15699.526} C_VEL
LIN {X 0,Y 340.491,Z 375.448,A -85,B 0,C 180,E1 15697.753,E2 15697.753} C_VEL
LIN {X 0,Y 334.422,Z 361.978,A -85,B 0,C 180,E1 15694.615,E2 15694.615} C_VEL
LIN {X 0,Y 328.952,Z 350.955,A -85,B 0,C 180,E1 15691.675,E2 15691.675} C_VEL
LIN {X 0,Y 324.536,Z 342.536,A -85,B 0,C 180,E1 15689.129,E2 15689.129} C_VEL
LIN {X 0,Y 321.981,Z 337.849,A -85,B 0,C 180,E1 15687.561,E2 15687.561} C_VEL
LIN {X 0,Y 319.574,Z 333.347,A -85,B 0,C 180,E1 15685.977,E2 15685.977} C_VEL
LIN {X 0,Y 317.442,Z 329.736,A -85,B 0,C 180,E1 15684.567,E2 15684.567} C_VEL
LIN {X 0,Y 316.736,Z 328.313,A -85,B 0,C 180,E1 15684.03,E2 15684.03} C_VEL
LIN {X 0,Y 314.637,Z 325.217,A -85,B 0,C 180,E1 15682.613,E2 15682.613} C_VEL
LIN {X 0,Y 314.147,Z 323.494,A -85,B 0,C 180,E1 15681.862,E2 15681.862} C_VEL
LIN {X 0,Y 314.123,Z 323.334,A -85,B 0,C 180,E1 15677.409,E2 15677.409} C_VEL
LIN {X 0,Y 314.129,Z 323.324,A -85,B 0,C 180,E1 15673.061,E2 15673.061} C_VEL
LIN {X 0,Y 314.146,Z 323.32,A -85,B 0,C 180,E1 15668.603,E2 15668.603} C_VEL
LIN {X 0,Y 314.126,Z 323.334,A -85,B 0,C 180,E1 15664.198,E2 15664.198} C_VEL
LIN {X 0,Y 314.109,Z 323.359,A -85,B 0,C 180,E1 15659.817,E2 15659.817} C_VEL
LIN {X 0,Y 314.103,Z 323.341,A -85,B 0,C 180,E1 15655.252,E2 15655.252} C_VEL
LIN {X 0,Y 314.117,Z 323.322,A -85,B 0,C 180,E1 15650.842,E2 15650.842} C_VEL
LIN {X 0,Y 314.146,Z 323.321,A -85,B 0,C 180,E1 15646.377,E2 15646.377} C_VEL
LIN {X 0,Y 314.139,Z 323.338,A -85,B 0,C 180,E1 15642.016,E2 15642.016} C_VEL
LIN {X 0,Y 314.126,Z 323.357,A -85,B 0,C 180,E1 15637.545,E2 15637.545} C_VEL
LIN {X 0,Y 314.129,Z 323.353,A -85,B 0,C 180,E1 15633.025,E2 15633.025} C_VEL
LIN {X 0,Y 314.161,Z 323.566,A -85,B 0,C 180,E1 15629.236,E2 15629.236} C_VEL
LIN {X 0,Y 315.946,Z 327.496,A -85,B 0,C 180,E1 15627.453,E2 15627.453} C_VEL
LIN {X 0,Y 316.972,Z 329.07,A -85,B 0,C 180,E1 15626.709,E2 15626.709} C_VEL
LIN {X 0,Y 318.886,Z 332.744,A -85,B 0,C 180,E1 15625.204,E2 15625.204} C_VEL
LIN {X 0,Y 321.869,Z 338.724,A -85,B 0,C 180,E1 15622.94,E2 15622.94} C_VEL
LIN {X 0,Y 325.849,Z 347.05,A -85,B 0,C 180,E1 15620.094,E2 15620.094} C_VEL
LIN {X 0,Y 328.116,Z 351.759,A -85,B 0,C 180,E1 15618.72,E2 15618.72} C_VEL
LIN {X 0,Y 337.734,Z 365.253,A -85,B 0,C 180,E1 15616.243,E2 15616.243} C_VEL
LIN {X 0,Y 347.005,Z 379.436,A -85,B 0,C 180,E1 15614.065,E2 15614.065} C_VEL
LIN {X 0,Y 356.673,Z 395.808,A -85,B 0,C 180,E1 15611.963,E2 15611.963} C_VEL
LIN {X 0,Y 359.573,Z 401.36,A -85,B 0,C 180,E1 15611.353,E2 15611.353} C_VEL
LIN {X 0,Y 353.247,Z 567.573,A -85,B 0,C 180,E1 15608.096,E2 15608.096} C_VEL
LIN {X 0,Y 352.129,Z 586.495,A -85,B 0,C 180,E1 15607.463,E2 15607.463} C_VEL
LIN {X 0,Y 350.278,Z 604.889,A -85,B 0,C 180,E1 15606.574,E2 15606.574} C_VEL
LIN {X 0,Y 347.767,Z 622.902,A -85,B 0,C 180,E1 15605.402,E2 15605.402} C_VEL
LIN {X 0,Y 344.698,Z 640.071,A -85,B 0,C 180,E1 15603.97,E2 15603.97} C_VEL
LIN {X 0,Y 341.125,Z 656.631,A -85,B 0,C 180,E1 15602.238,E2 15602.238} C_VEL
LIN {X 0,Y 337.325,Z 671.894,A -85,B 0,C 180,E1 15600.257,E2 15600.257} C_VEL
LIN {X 0,Y 333.507,Z 685.601,A -85,B 0,C 180,E1 15598.078,E2 15598.078} C_VEL
LIN {X 0,Y 329.534,Z 698.729,A -85,B 0,C 180,E1 15595.521,E2 15595.521} C_VEL
LIN {X 0,Y 325.815,Z 710.269,A -85,B 0,C 180,E1 15592.747,E2 15592.747} C_VEL
LIN {X 0,Y 322.507,Z 720.282,A -85,B 0,C 180,E1 15589.75,E2 15589.75} C_VEL
LIN {X 0,Y 319.671,Z 728.784,A -85,B 0,C 180,E1 15586.536,E2 15586.536} C_VEL
LIN {X 0,Y 317.426,Z 735.742,A -85,B 0,C 180,E1 15583.108,E2 15583.108} C_VEL
LIN {X 0,Y 315.876,Z 740.862,A -85,B 0,C 180,E1 15579.658,E2 15579.658} C_VEL
LIN {X 0,Y 314.856,Z 744.463,A -85,B 0,C 180,E1 15576.015,E2 15576.015} C_VEL
LIN {X 0,Y 314.374,Z 746.356,A -85,B 0,C 180,E1 15572.37,E2 15572.37} C_VEL
LIN {X 0,Y 314.307,Z 746.623,A -85,B 0,C 180,E1 15568.724,E2 15568.724} C_VEL
LIN {X 0,Y 314.648,Z 745.275,A -85,B 0,C 180,E1 15565.078,E2 15565.078} C_VEL
LIN {X 0,Y 315.483,Z 742.253,A -85,B 0,C 180,E1 15561.434,E2 15561.434} C_VEL
LIN {X 0,Y 316.827,Z 737.719,A -85,B 0,C 180,E1 15557.978,E2 15557.978} C_VEL
LIN {X 0,Y 318.828,Z 731.426,A -85,B 0,C 180,E1 15554.541,E2 15554.541} C_VEL
LIN {X 0,Y 321.426,Z 723.636,A -85,B 0,C 180,E1 15551.313,E2 15551.313} C_VEL
LIN {X 0,Y 324.492,Z 714.406,A -85,B 0,C 180,E1 15548.3,E2 15548.3} C_VEL
LIN {X 0,Y 327.978,Z 703.757,A -85,B 0,C 180,E1 15545.506,E2 15545.506} C_VEL
LIN {X 0,Y 331.759,Z 691.677,A -85,B 0,C 180,E1 15542.93,E2 15542.93} C_VEL
LIN {X 0,Y 334.7,Z 681.744,A -85,B 0,C 180,E1 15541.146,E2 15541.146} C_VEL
LIN {X 0,Y 335.348,Z 676.459,A -85,B 0,C 180,E1 15540.196,E2 15540.196} C_VEL
LIN {X 0,Y 334.122,Z 662.932,A -85,B 0,C 180,E1 15537.647,E2 15537.647} C_VEL
LIN {X 0,Y 334.618,Z 657.839,A -85,B 0,C 180,E1 15536.915,E2 15536.915} C_VEL
LIN {X 0,Y 334.817,Z 656.929,A -85,B 0,C 180,E1 15536.806,E2 15536.806} C_VEL
LIN {X 0,Y 338.568,Z 640.144,A -85,B 0,C 180,E1 15535.047,E2 15535.047} C_VEL
LIN {X 0,Y 341.814,Z 622.425,A -85,B 0,C 180,E1 15533.574,E2 15533.574} C_VEL
LIN {X 0,Y 344.345,Z 604.663,A -85,B 0,C 180,E1 15532.429,E2 15532.429} C_VEL
LIN {X 0,Y 346.287,Z 585.434,A -85,B 0,C 180,E1 15531.512,E2 15531.512} C_VEL
LIN {X 0,Y 347.4,Z 565.875,A -85,B 0,C 180,E1 15530.882,E2 15530.882} C_VEL
LIN {X 0,Y 353.769,Z 404.135,A -85,B 0,C 180,E1 15527.665,E2 15527.665} C_VEL
LIN {X 0,Y 343.89,Z 386.845,A -85,B 0,C 180,E1 15525.456,E2 15525.456} C_VEL
LIN {X 0,Y 334.213,Z 371.796,A -85,B 0,C 180,E1 15523.118,E2 15523.118} C_VEL
LIN {X 0,Y 325.345,Z 359.227,A -85,B 0,C 180,E1 15520.773,E2 15520.773} C_VEL
LIN {X 0,Y 319.968,Z 351.562,A -85,B 0,C 180,E1 15519.141,E2 15519.141} C_VEL
LIN {X 0,Y 315.753,Z 342.965,A -85,B 0,C 180,E1 15516.086,E2 15516.086} C_VEL
LIN {X 0,Y 313.3,Z 338.207,A -85,B 0,C 180,E1 15514.173,E2 15514.173} C_VEL
LIN {X 0,Y 311.037,Z 333.783,A -85,B 0,C 180,E1 15512.284,E2 15512.284} C_VEL
LIN {X 0,Y 309.082,Z 329.888,A -85,B 0,C 180,E1 15510.524,E2 15510.524} C_VEL
LIN {X 0,Y 306.478,Z 325.607,A -85,B 0,C 180,E1 15508.233,E2 15508.233} C_VEL
LIN {X 0,Y 306.221,Z 324.381,A -85,B 0,C 180,E1 15507.465,E2 15507.465} C_VEL
LIN {X 0,Y 306.189,Z 324.333,A -85,B 0,C 180,E1 15502.868,E2 15502.868} C_VEL
LIN {X 0,Y 306.19,Z 324.32,A -85,B 0,C 180,E1 15498.27,E2 15498.27} C_VEL
LIN {X 0,Y 306.21,Z 324.306,A -85,B 0,C 180,E1 15493.79,E2 15493.79} C_VEL
LIN {X 0,Y 306.195,Z 324.309,A -85,B 0,C 180,E1 15489.397,E2 15489.397} C_VEL
LIN {X 0,Y 306.18,Z 324.335,A -85,B 0,C 180,E1 15485.059,E2 15485.059} C_VEL
LIN {X 0,Y 306.163,Z 324.34,A -85,B 0,C 180,E1 15480.562,E2 15480.562} C_VEL
LIN {X 0,Y 306.17,Z 324.316,A -85,B 0,C 180,E1 15476.068,E2 15476.068} C_VEL
LIN {X 0,Y 306.194,Z 324.308,A -85,B 0,C 180,E1 15471.65,E2 15471.65} C_VEL
LIN {X 0,Y 306.201,Z 324.313,A -85,B 0,C 180,E1 15467.171,E2 15467.171} C_VEL
LIN {X 0,Y 306.187,Z 324.323,A -85,B 0,C 180,E1 15462.713,E2 15462.713} C_VEL
LIN {X 0,Y 306.245,Z 324.599,A -85,B 0,C 180,E1 15461.043,E2 15461.043} C_VEL
LIN {X 0,Y 307.653,Z 328.013,A -85,B 0,C 180,E1 15459.452,E2 15459.452} C_VEL
LIN {X 0,Y 309.466,Z 330.31,A -85,B 0,C 180,E1 15458.189,E2 15458.189} C_VEL
LIN {X 0,Y 311.515,Z 334.176,A -85,B 0,C 180,E1 15456.547,E2 15456.547} C_VEL
LIN {X 0,Y 312.362,Z 335.256,A -85,B 0,C 180,E1 15456.014,E2 15456.014} C_VEL
LIN {X 0,Y 314.296,Z 339.102,A -85,B 0,C 180,E1 15454.566,E2 15454.566} C_VEL
LIN {X 0,Y 315.38,Z 340.943,A -85,B 0,C 180,E1 15453.853,E2 15453.853} C_VEL
LIN {X 0,Y 318.179,Z 346.187,A -85,B 0,C 180,E1 15452.006,E2 15452.006} C_VEL
LIN {X 0,Y 322.463,Z 354.115,A -85,B 0,C 180,E1 15449.436,E2 15449.436} C_VEL
LIN {X 0,Y 328.196,Z 365.889,A -85,B 0,C 180,E1 15446.116,E2 15446.116} C_VEL
LIN {X 0,Y 332.812,Z 375.834,A -85,B 0,C 180,E1 15443.766,E2 15443.766} C_VEL
LIN {X 0,Y 342.739,Z 392.012,A -85,B 0,C 180,E1 15441.29,E2 15441.29} C_VEL
LIN {X 0,Y 351.771,Z 408.3,A -85,B 0,C 180,E1 15439.203,E2 15439.203} C_VEL
LIN {X 0,Y 352.815,Z 410.645,A -85,B 0,C 180,E1 15438.96,E2 15438.96} C_VEL
LIN {X 0,Y 354.231,Z 434.514,A -85,B 0,C 180,E1 15438.018,E2 15438.018} C_VEL
LIN {X 0,Y 344.514,Z 628.34,A -85,B 0,C 180,E1 15433.773,E2 15433.773} C_VEL
LIN {X 0,Y 342.227,Z 650.22,A -85,B 0,C 180,E1 15433.028,E2 15433.028} C_VEL
LIN {X 0,Y 338.992,Z 671.21,A -85,B 0,C 180,E1 15432.03,E2 15432.03} C_VEL
LIN {X 0,Y 335.114,Z 691.878,A -85,B 0,C 180,E1 15430.697,E2 15430.697} C_VEL
LIN {X 0,Y 330.856,Z 711.634,A -85,B 0,C 180,E1 15429.044,E2 15429.044} C_VEL
LIN {X 0,Y 326.287,Z 730.828,A -85,B 0,C 180,E1 15427.022,E2 15427.022} C_VEL
LIN {X 0,Y 321.717,Z 748.888,A -85,B 0,C 180,E1 15424.661,E2 15424.661} C_VEL
LIN {X 0,Y 317.37,Z 765.761,A -85,B 0,C 180,E1 15421.955,E2 15421.955} C_VEL
LIN {X 0,Y 313.494,Z 780.943,A -85,B 0,C 180,E1 15418.998,E2 15418.998} C_VEL
LIN {X 0,Y 310.269,Z 794.552,A -85,B 0,C 180,E1 15415.787,E2 15415.787} C_VEL
LIN {X 0,Y 307.763,Z 806.618,A -85,B 0,C 180,E1 15412.34,E2 15412.34} C_VEL
LIN {X 0,Y 306.12,Z 816.586,A -85,B 0,C 180,E1 15408.865,E2 15408.865} C_VEL
LIN {X 0,Y 305.216,Z 825.111,A -85,B 0,C 180,E1 15405.193,E2 15405.193} C_VEL
LIN {X 0,Y 304.956,Z 831.973,A -85,B 0,C 180,E1 15401.384,E2 15401.384} C_VEL
LIN {X 0,Y 305.136,Z 836.575,A -85,B 0,C 180,E1 15397.91,E2 15397.91} C_VEL
LIN {X 0,Y 305.456,Z 839.353,A -85,B 0,C 180,E1 15394.694,E2 15394.694} C_VEL
LIN {X 0,Y 305.688,Z 840.764,A -85,B 0,C 180,E1 15391.312,E2 15391.312} C_VEL
LIN {X 0,Y 305.669,Z 840.705,A -85,B 0,C 180,E1 15388.313,E2 15388.313} C_VEL
LIN {X 0,Y 305.426,Z 839.078,A -85,B 0,C 180,E1 15384.929,E2 15384.929} C_VEL
LIN {X 0,Y 305.094,Z 835.924,A -85,B 0,C 180,E1 15381.52,E2 15381.52} C_VEL
LIN {X 0,Y 304.952,Z 831.137,A -85,B 0,C 180,E1 15378.079,E2 15378.079} C_VEL
LIN {X 0,Y 305.247,Z 824.691,A -85,B 0,C 180,E1 15374.614,E2 15374.614} C_VEL
LIN {X 0,Y 306.194,Z 816.044,A -85,B 0,C 180,E1 15370.941,E2 15370.941} C_VEL
LIN {X 0,Y 307.879,Z 805.943,A -85,B 0,C 180,E1 15367.468,E2 15367.468} C_VEL
LIN {X 0,Y 310.267,Z 794.497,A -85,B 0,C 180,E1 15364.212,E2 15364.212} C_VEL
LIN {X 0,Y 313.489,Z 780.874,A -85,B 0,C 180,E1 15361.002,E2 15361.002} C_VEL
LIN {X 0,Y 317.364,Z 765.673,A -85,B 0,C 180,E1 15358.044,E2 15358.044} C_VEL
LIN {X 0,Y 321.709,Z 748.778,A -85,B 0,C 180,E1 15355.338,E2 15355.338} C_VEL
LIN {X 0,Y 326.277,Z 730.691,A -85,B 0,C 180,E1 15352.976,E2 15352.976} C_VEL
LIN {X 0,Y 330.824,Z 711.548,A -85,B 0,C 180,E1 15350.962,E2 15350.962} C_VEL
LIN {X 0,Y 334.859,Z 692.812,A -85,B 0,C 180,E1 15349.39,E2 15349.39} C_VEL
LIN {X 0,Y 338.64,Z 672.793,A -85,B 0,C 180,E1 15348.077,E2 15348.077} C_VEL
LIN {X 0,Y 341.824,Z 652.571,A -85,B 0,C 180,E1 15347.087,E2 15347.087} C_VEL
LIN {X 0,Y 344.13,Z 631.847,A -85,B 0,C 180,E1 15346.348,E2 15346.348} C_VEL
LIN {X 0,Y 345.878,Z 601.735,A -85,B 0,C 180,E1 15345.624,E2 15345.624} C_VEL
LIN {X 0,Y 354.16,Z 432.103,A -85,B 0,C 180,E1 15341.929,E2 15341.929} C_VEL
LIN {X 0,Y 352.517,Z 409.813,A -85,B 0,C 180,E1 15341.006,E2 15341.006} C_VEL
LIN {X 0,Y 342.98,Z 392.513,A -85,B 0,C 180,E1 15338.812,E2 15338.812} C_VEL
LIN {X 0,Y 332.766,Z 375.811,A -85,B 0,C 180,E1 15336.266,E2 15336.266} C_VEL
LIN {X 0,Y 327.862,Z 365.182,A -85,B 0,C 180,E1 15333.713,E2 15333.713} C_VEL
LIN {X 0,Y 322.081,Z 353.383,A -85,B 0,C 180,E1 15330.398,E2 15330.398} C_VEL
LIN {X 0,Y 317.199,Z 344.202,A -85,B 0,C 180,E1 15327.4,E2 15327.4} C_VEL
LIN {X 0,Y 314.49,Z 339.342,A -85,B 0,C 180,E1 15325.619,E2 15325.619} C_VEL
LIN {X 0,Y 312.477,Z 335.635,A -85,B 0,C 180,E1 15324.178,E2 15324.178} C_VEL
LIN {X 0,Y 309.559,Z 330.605,A -85,B 0,C 180,E1 15322.004,E2 15322.004} C_VEL
LIN {X 0,Y 308.589,Z 329.111,A -85,B 0,C 180,E1 15321.277,E2 15321.277} C_VEL
LIN {X 0,Y 306.537,Z 325.874,A -85,B 0,C 180,E1 15319.631,E2 15319.631} C_VEL
LIN {X 0,Y 306.22,Z 324.376,A -85,B 0,C 180,E1 15318.81,E2 15318.81} C_VEL
LIN {X 0,Y 306.203,Z 324.314,A -85,B 0,C 180,E1 15314.369,E2 15314.369} C_VEL
LIN {X 0,Y 306.182,Z 324.327,A -85,B 0,C 180,E1 15309.966,E2 15309.966} C_VEL
LIN {X 0,Y 306.172,Z 324.348,A -85,B 0,C 180,E1 15305.434,E2 15305.434} C_VEL
LIN {X 0,Y 306.18,Z 324.328,A -85,B 0,C 180,E1 15300.935,E2 15300.935} C_VEL
LIN {X 0,Y 306.186,Z 324.31,A -85,B 0,C 180,E1 15296.442,E2 15296.442} C_VEL
LIN {X 0,Y 306.188,Z 324.311,A -85,B 0,C 180,E1 15292.117,E2 15292.117} C_VEL
LIN {X 0,Y 306.171,Z 324.33,A -85,B 0,C 180,E1 15287.53,E2 15287.53} C_VEL
LIN {X 0,Y 306.179,Z 324.346,A -85,B 0,C 180,E1 15283.096,E2 15283.096} C_VEL
LIN {X 0,Y 306.205,Z 324.327,A -85,B 0,C 180,E1 15278.527,E2 15278.527} C_VEL
LIN {X 0,Y 306.212,Z 324.318,A -85,B 0,C 180,E1 15274.052,E2 15274.052} C_VEL
LIN {X 0,Y 306.262,Z 324.613,A -85,B 0,C 180,E1 15272.063,E2 15272.063} C_VEL
LIN {X 0,Y 307.646,Z 327.976,A -85,B 0,C 180,E1 15270.395,E2 15270.395} C_VEL
LIN {X 0,Y 309.101,Z 329.986,A -85,B 0,C 180,E1 15269.263,E2 15269.263} C_VEL
LIN {X 0,Y 311.029,Z 333.796,A -85,B 0,C 180,E1 15267.53,E2 15267.53} C_VEL
LIN {X 0,Y 312.131,Z 336.079,A -85,B 0,C 180,E1 15266.566,E2 15266.566} C_VEL
LIN {X 0,Y 314.327,Z 340.202,A -85,B 0,C 180,E1 15264.847,E2 15264.847} C_VEL
LIN {X 0,Y 316.781,Z 345.256,A -85,B 0,C 180,E1 15262.925,E2 15262.925} C_VEL
LIN {X 0,Y 320.44,Z 352.498,A -85,B 0,C 180,E1 15260.495,E2 15260.495} C_VEL
LIN {X 0,Y 331.091,Z 367.219,A -85,B 0,C 180,E1 15257.55,E2 15257.55} C_VEL
LIN {X 0,Y 340.99,Z 382.18,A -85,B 0,C 180,E1 15255.095,E2 15255.095} C_VEL
LIN {X 0,Y 351.296,Z 399.682,A -85,B 0,C 180,E1 15252.75,E2 15252.75} C_VEL
LIN {X 0,Y 353.779,Z 404.616,A -85,B 0,C 180,E1 15252.201,E2 15252.201} C_VEL
LIN {X 0,Y 347.238,Z 568.111,A -85,B 0,C 180,E1 15248.956,E2 15248.956} C_VEL
LIN {X 0,Y 346.071,Z 587.129,A -85,B 0,C 180,E1 15248.315,E2 15248.315} C_VEL
LIN {X 0,Y 344.189,Z 605.233,A -85,B 0,C 180,E1 15247.434,E2 15247.434} C_VEL
LIN {X 0,Y 341.573,Z 623.392,A -85,B 0,C 180,E1 15246.248,E2 15246.248} C_VEL
LIN {X 0,Y 338.33,Z 640.905,A -85,B 0,C 180,E1 15244.775,E2 15244.775} C_VEL
LIN {X 0,Y 334.605,Z 657.521,A -85,B 0,C 180,E1 15243.016,E2 15243.016} C_VEL
LIN {X 0,Y 330.694,Z 672.638,A -85,B 0,C 180,E1 15241.031,E2 15241.031} C_VEL
LIN {X 0,Y 326.556,Z 686.891,A -85,B 0,C 180,E1 15238.731,E2 15238.731} C_VEL
LIN {X 0,Y 322.412,Z 699.992,A -85,B 0,C 180,E1 15236.127,E2 15236.127} C_VEL
LIN {X 0,Y 318.524,Z 711.511,A -85,B 0,C 180,E1 15233.298,E2 15233.298} C_VEL
LIN {X 0,Y 315.056,Z 721.512,A -85,B 0,C 180,E1 15230.237,E2 15230.237} C_VEL
LIN {X 0,Y 312.075,Z 730.004,A -85,B 0,C 180,E1 15226.951,E2 15226.951} C_VEL
LIN {X 0,Y 309.705,Z 736.955,A -85,B 0,C 180,E1 15223.441,E2 15223.441} C_VEL
LIN {X 0,Y 308.066,Z 742.07,A -85,B 0,C 180,E1 15219.905,E2 15219.905} C_VEL
LIN {X 0,Y 306.982,Z 745.668,A -85,B 0,C 180,E1 15216.17,E2 15216.17} C_VEL
LIN {X 0,Y 306.47,Z 747.558,A -85,B 0,C 180,E1 15212.431,E2 15212.431} C_VEL
LIN {X 0,Y 306.399,Z 747.825,A -85,B 0,C 180,E1 15208.691,E2 15208.691} C_VEL
LIN {X 0,Y 306.762,Z 746.478,A -85,B 0,C 180,E1 15204.951,E2 15204.951} C_VEL
LIN {X 0,Y 307.649,Z 743.458,A -85,B 0,C 180,E1 15201.214,E2 15201.214} C_VEL
LIN {X 0,Y 309.073,Z 738.927,A -85,B 0,C 180,E1 15197.672,E2 15197.672} C_VEL
LIN {X 0,Y 311.188,Z 732.639,A -85,B 0,C 180,E1 15194.151,E2 15194.151} C_VEL
LIN {X 0,Y 313.922,Z 724.857,A -85,B 0,C 180,E1 15190.85,E2 15190.85} C_VEL
LIN {X 0,Y 317.14,Z 715.637,A -85,B 0,C 180,E1 15187.771,E2 15187.771} C_VEL
LIN {X 0,Y 320.789,Z 705.003,A -85,B 0,C 180,E1 15184.92,E2 15184.92} C_VEL
LIN {X 0,Y 324.736,Z 692.945,A -85,B 0,C 180,E1 15182.295,E2 15182.295} C_VEL
LIN {X 0,Y 328.847,Z 679.386,A -85,B 0,C 180,E1 15179.89,E2 15179.89} C_VEL
LIN {X 0,Y 333.022,Z 664.15,A -85,B 0,C 180,E1 15177.696,E2 15177.696} C_VEL
LIN {X 0,Y 334.817,Z 656.929,A -85,B 0,C 180,E1 15176.806,E2 15176.806} C_VEL
LIN {X 0,Y 335.517,Z 650.79,A -85,B 0,C 180,E1 15176.004,E2 15176.004} C_VEL
LIN {X 0,Y 334.288,Z 635.309,A -85,B 0,C 180,E1 15173.815,E2 15173.815} C_VEL
LIN {X 0,Y 334.729,Z 628.688,A -85,B 0,C 180,E1 15173.133,E2 15173.133} C_VEL
LIN {X 0,Y 337.61,Z 610.753,A -85,B 0,C 180,E1 15171.868,E2 15171.868} C_VEL
LIN {X 0,Y 339.875,Z 591.442,A -85,B 0,C 180,E1 15170.848,E2 15170.848} C_VEL
LIN {X 0,Y 341.288,Z 571.739,A -85,B 0,C 180,E1 15170.129,E2 15170.129} C_VEL
LIN {X 0,Y 343.314,Z 519.336,A -85,B 0,C 180,E1 15169.022,E2 15169.022} C_VEL
LIN {X 0,Y 348.016,Z 407.257,A -85,B 0,C 180,E1 15166.776,E2 15166.776} C_VEL
LIN {X 0,Y 338.565,Z 390.76,A -85,B 0,C 180,E1 15164.569,E2 15164.569} C_VEL
LIN {X 0,Y 329.597,Z 376.698,A -85,B 0,C 180,E1 15162.305,E2 15162.305} C_VEL
LIN {X 0,Y 320.047,Z 362.941,A -85,B 0,C 180,E1 15159.651,E2 15159.651} C_VEL
LIN {X 0,Y 312.328,Z 352.662,A -85,B 0,C 180,E1 15157.233,E2 15157.233} C_VEL
LIN {X 0,Y 309.703,Z 347.533,A -85,B 0,C 180,E1 15155.303,E2 15155.303} C_VEL
LIN {X 0,Y 308.074,Z 344.131,A -85,B 0,C 180,E1 15153.934,E2 15153.934} C_VEL
LIN {X 0,Y 305.835,Z 339.709,A -85,B 0,C 180,E1 15151.98,E2 15151.98} C_VEL
LIN {X 0,Y 303.526,Z 335.171,A -85,B 0,C 180,E1 15149.83,E2 15149.83} C_VEL
LIN {X 0,Y 301.465,Z 331.561,A -85,B 0,C 180,E1 15147.882,E2 15147.882} C_VEL
LIN {X 0,Y 300.708,Z 330.163,A -85,B 0,C 180,E1 15147.099,E2 15147.099} C_VEL
LIN {X 0,Y 298.483,Z 326.463,A -85,B 0,C 180,E1 15144.755,E2 15144.755} C_VEL
LIN {X 0,Y 298.286,Z 325.376,A -85,B 0,C 180,E1 15143.929,E2 15143.929} C_VEL
LIN {X 0,Y 298.261,Z 325.297,A -85,B 0,C 180,E1 15139.383,E2 15139.383} C_VEL
LIN {X 0,Y 298.242,Z 325.299,A -85,B 0,C 180,E1 15134.96,E2 15134.96} C_VEL
LIN {X 0,Y 298.241,Z 325.31,A -85,B 0,C 180,E1 15130.235,E2 15130.235} C_VEL
LIN {X 0,Y 298.257,Z 325.335,A -85,B 0,C 180,E1 15125.772,E2 15125.772} C_VEL
LIN {X 0,Y 298.241,Z 325.312,A -85,B 0,C 180,E1 15121.153,E2 15121.153} C_VEL
LIN {X 0,Y 298.226,Z 325.298,A -85,B 0,C 180,E1 15116.733,E2 15116.733} C_VEL
LIN {X 0,Y 298.233,Z 325.299,A -85,B 0,C 180,E1 15112.1,E2 15112.1} C_VEL
LIN {X 0,Y 298.258,Z 325.306,A -85,B 0,C 180,E1 15107.611,E2 15107.611} C_VEL
LIN {X 0,Y 298.273,Z 325.536,A -85,B 0,C 180,E1 15104.644,E2 15104.644} C_VEL
LIN {X 0,Y 300.103,Z 329.523,A -85,B 0,C 180,E1 15102.334,E2 15102.334} C_VEL
LIN {X 0,Y 301.545,Z 331.035,A -85,B 0,C 180,E1 15101.239,E2 15101.239} C_VEL
LIN {X 0,Y 303.231,Z 334.687,A -85,B 0,C 180,E1 15099.542,E2 15099.542} C_VEL
LIN {X 0,Y 304.739,Z 336.709,A -85,B 0,C 180,E1 15098.44,E2 15098.44} C_VEL
LIN {X 0,Y 307.091,Z 340.86,A -85,B 0,C 180,E1 15096.596,E2 15096.596} C_VEL
LIN {X 0,Y 310.57,Z 347.397,A -85,B 0,C 180,E1 15094.034,E2 15094.034} C_VEL
LIN {X 0,Y 313.239,Z 352.438,A -85,B 0,C 180,E1 15092.223,E2 15092.223} C_VEL
LIN {X 0,Y 317.212,Z 359.983,A -85,B 0,C 180,E1 15089.714,E2 15089.714} C_VEL
LIN {X 0,Y 322.945,Z 371.883,A -85,B 0,C 180,E1 15086.345,E2 15086.345} C_VEL
LIN {X 0,Y 324.709,Z 375.399,A -85,B 0,C 180,E1 15085.542,E2 15085.542} C_VEL
LIN {X 0,Y 334.641,Z 391.162,A -85,B 0,C 180,E1 15082.876,E2 15082.876} C_VEL
LIN {X 0,Y 343.495,Z 406.642,A -85,B 0,C 180,E1 15080.694,E2 15080.694} C_VEL
LIN {X 0,Y 347.369,Z 414.352,A -85,B 0,C 180,E1 15079.772,E2 15079.772} C_VEL
LIN {X 0,Y 348.511,Z 435.753,A -85,B 0,C 180,E1 15078.917,E2 15078.917} C_VEL
LIN {X 0,Y 338.522,Z 627.448,A -85,B 0,C 180,E1 15074.676,E2 15074.676} C_VEL
LIN {X 0,Y 336.163,Z 649.336,A -85,B 0,C 180,E1 15073.925,E2 15073.925} C_VEL
LIN {X 0,Y 332.862,Z 670.114,A -85,B 0,C 180,E1 15072.929,E2 15072.929} C_VEL
LIN {X 0,Y 328.796,Z 690.948,A -85,B 0,C 180,E1 15071.576,E2 15071.576} C_VEL
LIN {X 0,Y 324.522,Z 710.006,A -85,B 0,C 180,E1 15069.969,E2 15069.969} C_VEL
LIN {X 0,Y 319.911,Z 728.609,A -85,B 0,C 180,E1 15068.002,E2 15068.002} C_VEL
LIN {X 0,Y 315.591,Z 744.93,A -85,B 0,C 180,E1 15065.881,E2 15065.881} C_VEL
LIN {X 0,Y 311.177,Z 761.167,A -85,B 0,C 180,E1 15063.328,E2 15063.328} C_VEL
LIN {X 0,Y 307.169,Z 775.974,A -85,B 0,C 180,E1 15060.516,E2 15060.516} C_VEL
LIN {X 0,Y 303.504,Z 790.188,A -85,B 0,C 180,E1 15057.252,E2 15057.252} C_VEL
LIN {X 0,Y 300.59,Z 802.793,A -85,B 0,C 180,E1 15053.733,E2 15053.733} C_VEL
LIN {X 0,Y 298.623,Z 813.259,A -85,B 0,C 180,E1 15050.173,E2 15050.173} C_VEL
LIN {X 0,Y 297.44,Z 822.245,A -85,B 0,C 180,E1 15046.401,E2 15046.401} C_VEL
LIN {X 0,Y 296.992,Z 829.303,A -85,B 0,C 180,E1 15042.64,E2 15042.64} C_VEL
LIN {X 0,Y 297.099,Z 834.231,A -85,B 0,C 180,E1 15039.101,E2 15039.101} C_VEL
LIN {X 0,Y 297.429,Z 837.601,A -85,B 0,C 180,E1 15035.594,E2 15035.594} C_VEL
LIN {X 0,Y 297.723,Z 839.363,A -85,B 0,C 180,E1 15032.31,E2 15032.31} C_VEL
LIN {X 0,Y 297.792,Z 839.616,A -85,B 0,C 180,E1 15029.038,E2 15029.038} C_VEL
LIN {X 0,Y 297.566,Z 838.527,A -85,B 0,C 180,E1 15025.761,E2 15025.761} C_VEL
LIN {X 0,Y 297.233,Z 835.907,A -85,B 0,C 180,E1 15022.462,E2 15022.462} C_VEL
LIN {X 0,Y 296.994,Z 831.363,A -85,B 0,C 180,E1 15018.74,E2 15018.74} C_VEL
LIN {X 0,Y 297.205,Z 825.031,A -85,B 0,C 180,E1 15014.987,E2 15014.987} C_VEL
LIN {X 0,Y 298.078,Z 816.808,A -85,B 0,C 180,E1 15011.216,E2 15011.216} C_VEL
LIN {X 0,Y 299.838,Z 806.52,A -85,B 0,C 180,E1 15007.451,E2 15007.451} C_VEL
LIN {X 0,Y 302.426,Z 794.641,A -85,B 0,C 180,E1 15003.915,E2 15003.915} C_VEL
LIN {X 0,Y 305.758,Z 781.237,A -85,B 0,C 180,E1 15000.627,E2 15000.627} C_VEL
LIN {X 0,Y 309.764,Z 766.307,A -85,B 0,C 180,E1 14997.602,E2 14997.602} C_VEL
LIN {X 0,Y 313.918,Z 750.922,A -85,B 0,C 180,E1 14995.019,E2 14995.019} C_VEL
LIN {X 0,Y 318.404,Z 734.168,A -85,B 0,C 180,E1 14992.696,E2 14992.696} C_VEL
LIN {X 0,Y 323.05,Z 715.791,A -85,B 0,C 180,E1 14990.619,E2 14990.619} C_VEL
LIN {X 0,Y 327.542,Z 696.359,A -85,B 0,C 180,E1 14988.866,E2 14988.866} C_VEL
LIN {X 0,Y 331.503,Z 677.008,A -85,B 0,C 180,E1 14987.5,E2 14987.5} C_VEL
LIN {X 0,Y 334.931,Z 657.164,A -85,B 0,C 180,E1 14986.433,E2 14986.433} C_VEL
LIN {X 0,Y 337.6,Z 636.588,A -85,B 0,C 180,E1 14985.621,E2 14985.621} C_VEL
LIN {X 0,Y 339.243,Z 614.759,A -85,B 0,C 180,E1 14985.024,E2 14985.024} C_VEL
LIN {X 0,Y 348.464,Z 433.38,A -85,B 0,C 180,E1 14981.034,E2 14981.034} C_VEL
LIN {X 0,Y 347.056,Z 413.552,A -85,B 0,C 180,E1 14980.191,E2 14980.191} C_VEL
LIN {X 0,Y 338.3,Z 397.503,A -85,B 0,C 180,E1 14978.095,E2 14978.095} C_VEL
LIN {X 0,Y 328.678,Z 381.539,A -85,B 0,C 180,E1 14975.603,E2 14975.603} C_VEL
LIN {X 0,Y 323.71,Z 373.599,A -85,B 0,C 180,E1 14974.131,E2 14974.131} C_VEL
LIN {X 0,Y 318.309,Z 362.299,A -85,B 0,C 180,E1 14971.007,E2 14971.007} C_VEL
LIN {X 0,Y 313.987,Z 353.863,A -85,B 0,C 180,E1 14968.325,E2 14968.325} C_VEL
LIN {X 0,Y 311.504,Z 349.228,A -85,B 0,C 180,E1 14966.703,E2 14966.703} C_VEL
LIN {X 0,Y 309.417,Z 345.303,A -85,B 0,C 180,E1 14965.248,E2 14965.248} C_VEL
LIN {X 0,Y 306.965,Z 340.727,A -85,B 0,C 180,E1 14963.414,E2 14963.414} C_VEL
LIN {X 0,Y 304.831,Z 336.987,A -85,B 0,C 180,E1 14961.755,E2 14961.755} C_VEL
LIN {X 0,Y 303.891,Z 335.482,A -85,B 0,C 180,E1 14961.016,E2 14961.016} C_VEL
LIN {X 0,Y 301.737,Z 331.756,A -85,B 0,C 180,E1 14959.15,E2 14959.15} C_VEL
LIN {X 0,Y 300.935,Z 330.339,A -85,B 0,C 180,E1 14958.399,E2 14958.399} C_VEL
LIN {X 0,Y 298.671,Z 327.035,A -85,B 0,C 180,E1 14956.332,E2 14956.332} C_VEL
LIN {X 0,Y 298.264,Z 325.446,A -85,B 0,C 180,E1 14955.356,E2 14955.356} C_VEL
LIN {X 0,Y 298.261,Z 325.333,A -85,B 0,C 180,E1 14950.82,E2 14950.82} C_VEL
LIN {X 0,Y 298.26,Z 325.316,A -85,B 0,C 180,E1 14946.351,E2 14946.351} C_VEL
LIN {X 0,Y 298.227,Z 325.305,A -85,B 0,C 180,E1 14941.729,E2 14941.729} C_VEL
LIN {X 0,Y 298.225,Z 325.298,A -85,B 0,C 180,E1 14937.117,E2 14937.117} C_VEL
LIN {X 0,Y 298.248,Z 325.305,A -85,B 0,C 180,E1 14932.681,E2 14932.681} C_VEL
LIN {X 0,Y 298.258,Z 325.33,A -85,B 0,C 180,E1 14928.196,E2 14928.196} C_VEL
LIN {X 0,Y 298.244,Z 325.321,A -85,B 0,C 180,E1 14923.643,E2 14923.643} C_VEL
LIN {X 0,Y 298.245,Z 325.309,A -85,B 0,C 180,E1 14918.978,E2 14918.978} C_VEL
LIN {X 0,Y 298.291,Z 325.596,A -85,B 0,C 180,E1 14915.545,E2 14915.545} C_VEL
LIN {X 0,Y 300.232,Z 329.679,A -85,B 0,C 180,E1 14913.068,E2 14913.068} C_VEL
LIN {X 0,Y 301.324,Z 331.131,A -85,B 0,C 180,E1 14912.104,E2 14912.104} C_VEL
LIN {X 0,Y 303.026,Z 334.6,A -85,B 0,C 180,E1 14910.334,E2 14910.334} C_VEL
LIN {X 0,Y 304.139,Z 336.451,A -85,B 0,C 180,E1 14909.365,E2 14909.365} C_VEL
LIN {X 0,Y 306.759,Z 341.521,A -85,B 0,C 180,E1 14907.021,E2 14907.021} C_VEL
LIN {X 0,Y 309.09,Z 346.172,A -85,B 0,C 180,E1 14905.07,E2 14905.07} C_VEL
LIN {X 0,Y 312.683,Z 353.174,A -85,B 0,C 180,E1 14902.467,E2 14902.467} C_VEL
LIN {X 0,Y 321.163,Z 364.628,A -85,B 0,C 180,E1 14899.876,E2 14899.876} C_VEL
LIN {X 0,Y 330.578,Z 378.201,A -85,B 0,C 180,E1 14897.303,E2 14897.303} C_VEL
LIN {X 0,Y 340.215,Z 393.56,A -85,B 0,C 180,E1 14894.905,E2 14894.905} C_VEL
LIN {X 0,Y 348.072,Z 407.676,A -85,B 0,C 180,E1 14893.08,E2 14893.08} C_VEL
LIN {X 0,Y 341.306,Z 568.746,A -85,B 0,C 180,E1 14889.843,E2 14889.843} C_VEL
LIN {X 0,Y 340.081,Z 587.888,A -85,B 0,C 180,E1 14889.191,E2 14889.191} C_VEL
LIN {X 0,Y 338.085,Z 606.306,A -85,B 0,C 180,E1 14888.284,E2 14888.284} C_VEL
LIN {X 0,Y 335.455,Z 623.878,A -85,B 0,C 180,E1 14887.125,E2 14887.125} C_VEL
LIN {X 0,Y 332.137,Z 641.248,A -85,B 0,C 180,E1 14885.656,E2 14885.656} C_VEL
LIN {X 0,Y 328.255,Z 657.979,A -85,B 0,C 180,E1 14883.876,E2 14883.876} C_VEL
LIN {X 0,Y 324.125,Z 673.382,A -85,B 0,C 180,E1 14881.836,E2 14881.836} C_VEL
LIN {X 0,Y 319.951,Z 687.213,A -85,B 0,C 180,E1 14879.587,E2 14879.587} C_VEL
LIN {X 0,Y 315.6,Z 700.452,A -85,B 0,C 180,E1 14876.938,E2 14876.938} C_VEL
LIN {X 0,Y 311.501,Z 712.095,A -85,B 0,C 180,E1 14874.056,E2 14874.056} C_VEL
LIN {X 0,Y 307.822,Z 722.207,A -85,B 0,C 180,E1 14870.934,E2 14870.934} C_VEL
LIN {X 0,Y 304.651,Z 730.8,A -85,B 0,C 180,E1 14867.574,E2 14867.574} C_VEL
LIN {X 0,Y 302.105,Z 737.845,A -85,B 0,C 180,E1 14863.981,E2 14863.981} C_VEL
LIN {X 0,Y 300.335,Z 743.048,A -85,B 0,C 180,E1 14860.356,E2 14860.356} C_VEL
LIN {X 0,Y 299.151,Z 746.729,A -85,B 0,C 180,E1 14856.525,E2 14856.525} C_VEL
LIN {X 0,Y 298.579,Z 748.7,A -85,B 0,C 180,E1 14852.687,E2 14852.687} C_VEL
LIN {X 0,Y 298.487,Z 749.045,A -85,B 0,C 180,E1 14848.848,E2 14848.848} C_VEL
LIN {X 0,Y 298.845,Z 747.781,A -85,B 0,C 180,E1 14845.01,E2 14845.01} C_VEL
LIN {X 0,Y 299.756,Z 744.849,A -85,B 0,C 180,E1 14841.174,E2 14841.174} C_VEL
LIN {X 0,Y 301.233,Z 740.412,A -85,B 0,C 180,E1 14837.541,E2 14837.541} C_VEL
LIN {X 0,Y 303.425,Z 734.224,A -85,B 0,C 180,E1 14833.931,E2 14833.931} C_VEL
LIN {X 0,Y 306.26,Z 726.554,A -85,B 0,C 180,E1 14830.549,E2 14830.549} C_VEL
LIN {X 0,Y 309.598,Z 717.462,A -85,B 0,C 180,E1 14827.399,E2 14827.399} C_VEL
LIN {X 0,Y 313.635,Z 706.249,A -85,B 0,C 180,E1 14824.307,E2 14824.307} C_VEL
LIN {X 0,Y 317.755,Z 694.212,A -85,B 0,C 180,E1 14821.632,E2 14821.632} C_VEL
LIN {X 0,Y 322.118,Z 680.418,A -85,B 0,C 180,E1 14819.141,E2 14819.141} C_VEL
LIN {X 0,Y 326.383,Z 665.492,A -85,B 0,C 180,E1 14816.956,E2 14816.956} C_VEL
LIN {X 0,Y 330.298,Z 649.867,A -85,B 0,C 180,E1 14815.102,E2 14815.102} C_VEL
LIN {X 0,Y 334.018,Z 632.337,A -85,B 0,C 180,E1 14813.439,E2 14813.439} C_VEL
LIN {X 0,Y 334.729,Z 628.688,A -85,B 0,C 180,E1 14813.133,E2 14813.133} C_VEL
LIN {X 0,Y 335.223,Z 621.912,A -85,B 0,C 180,E1 14812.488,E2 14812.488} C_VEL
LIN {X 0,Y 333.336,Z 605.824,A -85,B 0,C 180,E1 14810.785,E2 14810.785} C_VEL
LIN {X 0,Y 333.268,Z 598.698,A -85,B 0,C 180,E1 14810.261,E2 14810.261} C_VEL
LIN {X 0,Y 333.358,Z 597.642,A -85,B 0,C 180,E1 14810.205,E2 14810.205} C_VEL
LIN {X 0,Y 335.063,Z 578.214,A -85,B 0,C 180,E1 14809.399,E2 14809.399} C_VEL
LIN {X 0,Y 336.115,Z 554.132,A -85,B 0,C 180,E1 14808.778,E2 14808.778} C_VEL
LIN {X 0,Y 342.447,Z 410.601,A -85,B 0,C 180,E1 14805.881,E2 14805.881} C_VEL
LIN {X 0,Y 332.833,Z 393.769,A -85,B 0,C 180,E1 14803.527,E2 14803.527} C_VEL
LIN {X 0,Y 323.264,Z 378.915,A -85,B 0,C 180,E1 14800.975,E2 14800.975} C_VEL
LIN {X 0,Y 313.207,Z 364.634,A -85,B 0,C 180,E1 14797.976,E2 14797.976} C_VEL
LIN {X 0,Y 304.622,Z 353.575,A -85,B 0,C 180,E1 14795.058,E2 14795.058} C_VEL
LIN {X 0,Y 302.664,Z 349.691,A -85,B 0,C 180,E1 14793.483,E2 14793.483} C_VEL
LIN {X 0,Y 300.659,Z 345.658,A -85,B 0,C 180,E1 14791.698,E2 14791.698} C_VEL
LIN {X 0,Y 298.421,Z 341.198,A -85,B 0,C 180,E1 14789.507,E2 14789.507} C_VEL
LIN {X 0,Y 296.48,Z 337.511,A -85,B 0,C 180,E1 14787.511,E2 14787.511} C_VEL
LIN {X 0,Y 293.618,Z 332.441,A -85,B 0,C 180,E1 14784.334,E2 14784.334} C_VEL
LIN {X 0,Y 292.341,Z 330.711,A -85,B 0,C 180,E1 14782.949,E2 14782.949} C_VEL
LIN {X 0,Y 290.377,Z 326.58,A -85,B 0,C 180,E1 14779.722,E2 14779.722} C_VEL
LIN {X 0,Y 290.32,Z 326.289,A -85,B 0,C 180,E1 14775.358,E2 14775.358} C_VEL
LIN {X 0,Y 290.297,Z 326.308,A -85,B 0,C 180,E1 14770.719,E2 14770.719} C_VEL
LIN {X 0,Y 290.301,Z 326.318,A -85,B 0,C 180,E1 14766.13,E2 14766.13} C_VEL
LIN {X 0,Y 290.313,Z 326.291,A -85,B 0,C 180,E1 14761.579,E2 14761.579} C_VEL
LIN {X 0,Y 290.297,Z 326.283,A -85,B 0,C 180,E1 14757.039,E2 14757.039} C_VEL
LIN {X 0,Y 290.29,Z 326.29,A -85,B 0,C 180,E1 14752.48,E2 14752.48} C_VEL
LIN {X 0,Y 290.362,Z 326.628,A -85,B 0,C 180,E1 14749.083,E2 14749.083} C_VEL
LIN {X 0,Y 292.426,Z 330.794,A -85,B 0,C 180,E1 14745.951,E2 14745.951} C_VEL
LIN {X 0,Y 293.803,Z 332.415,A -85,B 0,C 180,E1 14744.607,E2 14744.607} C_VEL
LIN {X 0,Y 295.909,Z 336.401,A -85,B 0,C 180,E1 14742.296,E2 14742.296} C_VEL
LIN {X 0,Y 296.9,Z 337.395,A -85,B 0,C 180,E1 14741.545,E2 14741.545} C_VEL
LIN {X 0,Y 298.811,Z 341.358,A -85,B 0,C 180,E1 14739.636,E2 14739.636} C_VEL
LIN {X 0,Y 300.03,Z 343.088,A -85,B 0,C 180,E1 14738.701,E2 14738.701} C_VEL
LIN {X 0,Y 303.003,Z 348.659,A -85,B 0,C 180,E1 14736.261,E2 14736.261} C_VEL
LIN {X 0,Y 305.756,Z 353.796,A -85,B 0,C 180,E1 14734.22,E2 14734.22} C_VEL
LIN {X 0,Y 309.863,Z 361.613,A -85,B 0,C 180,E1 14731.361,E2 14731.361} C_VEL
LIN {X 0,Y 315.892,Z 373.809,A -85,B 0,C 180,E1 14727.716,E2 14727.716} C_VEL
LIN {X 0,Y 324.972,Z 387.721,A -85,B 0,C 180,E1 14725.038,E2 14725.038} C_VEL
LIN {X 0,Y 334.512,Z 403.802,A -85,B 0,C 180,E1 14722.482,E2 14722.482} C_VEL
LIN {X 0,Y 341.977,Z 417.8,A -85,B 0,C 180,E1 14720.621,E2 14720.621} C_VEL
LIN {X 0,Y 342.894,Z 436.769,A -85,B 0,C 180,E1 14719.85,E2 14719.85} C_VEL
LIN {X 0,Y 332.625,Z 626.475,A -85,B 0,C 180,E1 14715.614,E2 14715.614} C_VEL
LIN {X 0,Y 330.213,Z 648.278,A -85,B 0,C 180,E1 14714.861,E2 14714.861} C_VEL
LIN {X 0,Y 326.821,Z 669.02,A -85,B 0,C 180,E1 14713.862,E2 14713.862} C_VEL
LIN {X 0,Y 322.839,Z 688.695,A -85,B 0,C 180,E1 14712.586,E2 14712.586} C_VEL
LIN {X 0,Y 318.472,Z 707.543,A -85,B 0,C 180,E1 14711.007,E2 14711.007} C_VEL
LIN {X 0,Y 313.842,Z 725.625,A -85,B 0,C 180,E1 14709.108,E2 14709.108} C_VEL
LIN {X 0,Y 309.037,Z 743.042,A -85,B 0,C 180,E1 14706.852,E2 14706.852} C_VEL
LIN {X 0,Y 304.41,Z 759.264,A -85,B 0,C 180,E1 14704.284,E2 14704.284} C_VEL
LIN {X 0,Y 300.01,Z 774.636,A -85,B 0,C 180,E1 14701.325,E2 14701.325} C_VEL
LIN {X 0,Y 296.308,Z 788.111,A -85,B 0,C 180,E1 14698.19,E2 14698.19} C_VEL
LIN {X 0,Y 293.28,Z 800.234,A -85,B 0,C 180,E1 14694.792,E2 14694.792} C_VEL
LIN {X 0,Y 291.041,Z 810.954,A -85,B 0,C 180,E1 14691.144,E2 14691.144} C_VEL
LIN {X 0,Y 289.627,Z 820.148,A -85,B 0,C 180,E1 14687.27,E2 14687.27} C_VEL
LIN {X 0,Y 289.057,Z 827.365,A -85,B 0,C 180,E1 14683.4,E2 14683.4} C_VEL
LIN {X 0,Y 289.113,Z 832.759,A -85,B 0,C 180,E1 14679.555,E2 14679.555} C_VEL
LIN {X 0,Y 289.472,Z 836.309,A -85,B 0,C 180,E1 14675.863,E2 14675.863} C_VEL
LIN {X 0,Y 289.794,Z 838.08,A -85,B 0,C 180,E1 14672.571,E2 14672.571} C_VEL
LIN {X 0,Y 289.886,Z 838.441,A -85,B 0,C 180,E1 14669.209,E2 14669.209} C_VEL
LIN {X 0,Y 289.668,Z 837.477,A -85,B 0,C 180,E1 14665.987,E2 14665.987} C_VEL
LIN {X 0,Y 289.291,Z 834.873,A -85,B 0,C 180,E1 14662.453,E2 14662.453} C_VEL
LIN {X 0,Y 289.03,Z 830.708,A -85,B 0,C 180,E1 14658.83,E2 14658.83} C_VEL
LIN {X 0,Y 289.219,Z 824.56,A -85,B 0,C 180,E1 14654.973,E2 14654.973} C_VEL
LIN {X 0,Y 290.106,Z 816.47,A -85,B 0,C 180,E1 14651.097,E2 14651.097} C_VEL
LIN {X 0,Y 291.797,Z 806.944,A -85,B 0,C 180,E1 14647.433,E2 14647.433} C_VEL
LIN {X 0,Y 294.417,Z 795.415,A -85,B 0,C 180,E1 14643.802,E2 14643.802} C_VEL
LIN {X 0,Y 297.853,Z 782.251,A -85,B 0,C 180,E1 14640.392,E2 14640.392} C_VEL
LIN {X 0,Y 302.056,Z 767.37,A -85,B 0,C 180,E1 14637.222,E2 14637.222} C_VEL
LIN {X 0,Y 306.64,Z 751.293,A -85,B 0,C 180,E1 14634.408,E2 14634.408} C_VEL
LIN {X 0,Y 311.475,Z 734.13,A -85,B 0,C 180,E1 14631.952,E2 14631.952} C_VEL
LIN {X 0,Y 316.088,Z 716.815,A -85,B 0,C 180,E1 14629.932,E2 14629.932} C_VEL
LIN {X 0,Y 320.628,Z 698.246,A -85,B 0,C 180,E1 14628.185,E2 14628.185} C_VEL
LIN {X 0,Y 324.793,Z 679.161,A -85,B 0,C 180,E1 14626.769,E2 14626.769} C_VEL
LIN {X 0,Y 328.496,Z 659.002,A -85,B 0,C 180,E1 14625.631,E2 14625.631} C_VEL
LIN {X 0,Y 331.501,Z 637.353,A -85,B 0,C 180,E1 14624.742,E2 14624.742} C_VEL
LIN {X 0,Y 333.284,Z 615.358,A -85,B 0,C 180,E1 14624.119,E2 14624.119} C_VEL
LIN {X 0,Y 342.847,Z 434.463,A -85,B 0,C 180,E1 14620.101,E2 14620.101} C_VEL
LIN {X 0,Y 341.646,Z 417.212,A -85,B 0,C 180,E1 14619.343,E2 14619.343} C_VEL
LIN {X 0,Y 332.368,Z 400.123,A -85,B 0,C 180,E1 14617.015,E2 14617.015} C_VEL
LIN {X 0,Y 323.108,Z 384.877,A -85,B 0,C 180,E1 14614.492,E2 14614.492} C_VEL
LIN {X 0,Y 315.51,Z 373.117,A -85,B 0,C 180,E1 14612.167,E2 14612.167} C_VEL
LIN {X 0,Y 309.723,Z 361.189,A -85,B 0,C 180,E1 14608.54,E2 14608.54} C_VEL
LIN {X 0,Y 304.664,Z 351.646,A -85,B 0,C 180,E1 14605.046,E2 14605.046} C_VEL
LIN {X 0,Y 301.904,Z 346.675,A -85,B 0,C 180,E1 14602.976,E2 14602.976} C_VEL
LIN {X 0,Y 299.449,Z 342.125,A -85,B 0,C 180,E1 14600.932,E2 14600.932} C_VEL
LIN {X 0,Y 297.074,Z 338.101,A -85,B 0,C 180,E1 14598.85,E2 14598.85} C_VEL
LIN {X 0,Y 296.51,Z 336.975,A -85,B 0,C 180,E1 14598.276,E2 14598.276} C_VEL
LIN {X 0,Y 294.245,Z 333.717,A -85,B 0,C 180,E1 14596.179,E2 14596.179} C_VEL
LIN {X 0,Y 293.336,Z 331.648,A -85,B 0,C 180,E1 14595.013,E2 14595.013} C_VEL
LIN {X 0,Y 290.735,Z 328.06,A -85,B 0,C 180,E1 14592.109,E2 14592.109} C_VEL
LIN {X 0,Y 290.339,Z 326.466,A -85,B 0,C 180,E1 14590.918,E2 14590.918} C_VEL
LIN {X 0,Y 290.33,Z 326.299,A -85,B 0,C 180,E1 14586.525,E2 14586.525} C_VEL
LIN {X 0,Y 290.295,Z 326.289,A -85,B 0,C 180,E1 14581.973,E2 14581.973} C_VEL
LIN {X 0,Y 290.281,Z 326.288,A -85,B 0,C 180,E1 14577.433,E2 14577.433} C_VEL
LIN {X 0,Y 290.299,Z 326.298,A -85,B 0,C 180,E1 14572.877,E2 14572.877} C_VEL
LIN {X 0,Y 290.32,Z 326.319,A -85,B 0,C 180,E1 14568.276,E2 14568.276} C_VEL
LIN {X 0,Y 290.31,Z 326.304,A -85,B 0,C 180,E1 14563.801,E2 14563.801} C_VEL
LIN {X 0,Y 290.365,Z 326.591,A -85,B 0,C 180,E1 14559.973,E2 14559.973} C_VEL
LIN {X 0,Y 292.309,Z 330.67,A -85,B 0,C 180,E1 14556.836,E2 14556.836} C_VEL
LIN {X 0,Y 293.589,Z 332.42,A -85,B 0,C 180,E1 14555.449,E2 14555.449} C_VEL
LIN {X 0,Y 295.674,Z 336.283,A -85,B 0,C 180,E1 14553.054,E2 14553.054} C_VEL
LIN {X 0,Y 296.465,Z 337.573,A -85,B 0,C 180,E1 14552.262,E2 14552.262} C_VEL
LIN {X 0,Y 298.639,Z 341.479,A -85,B 0,C 180,E1 14550.126,E2 14550.126} C_VEL
LIN {X 0,Y 301.629,Z 347.502,A -85,B 0,C 180,E1 14547.294,E2 14547.294} C_VEL
LIN {X 0,Y 304.135,Z 352.694,A -85,B 0,C 180,E1 14545.107,E2 14545.107} C_VEL
LIN {X 0,Y 306.245,Z 355.597,A -85,B 0,C 180,E1 14544.18,E2 14544.18} C_VEL
LIN {X 0,Y 314.388,Z 366.42,A -85,B 0,C 180,E1 14541.497,E2 14541.497} C_VEL
LIN {X 0,Y 323.76,Z 379.679,A -85,B 0,C 180,E1 14538.749,E2 14538.749} C_VEL
LIN {X 0,Y 333.437,Z 394.86,A -85,B 0,C 180,E1 14536.186,E2 14536.186} C_VEL
LIN {X 0,Y 342.449,Z 410.811,A -85,B 0,C 180,E1 14533.988,E2 14533.988} C_VEL
LIN {X 0,Y 335.457,Z 569.4,A -85,B 0,C 180,E1 14530.76,E2 14530.76} C_VEL
LIN {X 0,Y 334.185,Z 588.515,A -85,B 0,C 180,E1 14530.104,E2 14530.104} C_VEL
LIN {X 0,Y 332.059,Z 607.376,A -85,B 0,C 180,E1 14529.165,E2 14529.165} C_VEL
LIN {X 0,Y 329.274,Z 625.188,A -85,B 0,C 180,E1 14527.971,E2 14527.971} C_VEL
LIN {X 0,Y 325.721,Z 642.956,A -85,B 0,C 180,E1 14526.439,E2 14526.439} C_VEL
LIN {X 0,Y 321.742,Z 659.358,A -85,B 0,C 180,E1 14524.658,E2 14524.658} C_VEL
LIN {X 0,Y 317.359,Z 675.002,A -85,B 0,C 180,E1 14522.543,E2 14522.543} C_VEL
LIN {X 0,Y 313.103,Z 688.498,A -85,B 0,C 180,E1 14520.301,E2 14520.301} C_VEL
LIN {X 0,Y 308.567,Z 701.711,A -85,B 0,C 180,E1 14517.604,E2 14517.604} C_VEL
LIN {X 0,Y 304.284,Z 713.336,A -85,B 0,C 180,E1 14514.664,E2 14514.664} C_VEL
LIN {X 0,Y 300.429,Z 723.435,A -85,B 0,C 180,E1 14511.474,E2 14511.474} C_VEL
LIN {X 0,Y 297.099,Z 732.018,A -85,B 0,C 180,E1 14508.036,E2 14508.036} C_VEL
LIN {X 0,Y 294.413,Z 739.058,A -85,B 0,C 180,E1 14504.354,E2 14504.354} C_VEL
LIN {X 0,Y 292.54,Z 744.256,A -85,B 0,C 180,E1 14500.635,E2 14500.635} C_VEL
LIN {X 0,Y 291.285,Z 747.933,A -85,B 0,C 180,E1 14496.702,E2 14496.702} C_VEL
LIN {X 0,Y 290.676,Z 749.902,A -85,B 0,C 180,E1 14492.76,E2 14492.76} C_VEL
LIN {X 0,Y 290.578,Z 750.247,A -85,B 0,C 180,E1 14488.817,E2 14488.817} C_VEL
LIN {X 0,Y 290.961,Z 748.983,A -85,B 0,C 180,E1 14484.874,E2 14484.874} C_VEL
LIN {X 0,Y 291.928,Z 746.053,A -85,B 0,C 180,E1 14480.936,E2 14480.936} C_VEL
LIN {X 0,Y 293.492,Z 741.62,A -85,B 0,C 180,E1 14477.207,E2 14477.207} C_VEL
LIN {X 0,Y 295.809,Z 735.438,A -85,B 0,C 180,E1 14473.506,E2 14473.506} C_VEL
LIN {X 0,Y 298.793,Z 727.774,A -85,B 0,C 180,E1 14470.043,E2 14470.043} C_VEL
LIN {X 0,Y 302.523,Z 718.097,A -85,B 0,C 180,E1 14466.634,E2 14466.634} C_VEL
LIN {X 0,Y 306.519,Z 707.492,A -85,B 0,C 180,E1 14463.665,E2 14463.665} C_VEL
LIN {X 0,Y 310.818,Z 695.477,A -85,B 0,C 180,E1 14460.94,E2 14460.94} C_VEL
LIN {X 0,Y 315.28,Z 681.98,A -85,B 0,C 180,E1 14458.449,E2 14458.449} C_VEL
LIN {X 0,Y 319.801,Z 666.833,A -85,B 0,C 180,E1 14456.186,E2 14456.186} C_VEL
LIN {X 0,Y 324.039,Z 650.566,A -85,B 0,C 180,E1 14454.229,E2 14454.229} C_VEL
LIN {X 0,Y 327.734,Z 633.843,A -85,B 0,C 180,E1 14452.62,E2 14452.62} C_VEL
LIN {X 0,Y 330.992,Z 615.43,A -85,B 0,C 180,E1 14451.228,E2 14451.228} C_VEL
LIN {X 0,Y 333.358,Z 597.642,A -85,B 0,C 180,E1 14450.205,E2 14450.205} C_VEL
LIN {X 0,Y 333.417,Z 590.341,A -85,B 0,C 180,E1 14449.748,E2 14449.748} C_VEL
LIN {X 0,Y 330.472,Z 572.138,A -85,B 0,C 180,E1 14448.365,E2 14448.365} C_VEL
LIN {X 0,Y 330.034,Z 564.642,A -85,B 0,C 180,E1 14448.039,E2 14448.039} C_VEL
LIN {X 0,Y 336.89,Z 413.857,A -85,B 0,C 180,E1 14444.94,E2 14444.94} C_VEL
LIN {X 0,Y 327.682,Z 397.794,A -85,B 0,C 180,E1 14442.581,E2 14442.581} C_VEL
LIN {X 0,Y 318.487,Z 383.339,A -85,B 0,C 180,E1 14440.005,E2 14440.005} C_VEL
LIN {X 0,Y 309.533,Z 370.652,A -85,B 0,C 180,E1 14437.219,E2 14437.219} C_VEL
LIN {X 0,Y 302.01,Z 360.764,A -85,B 0,C 180,E1 14434.596,E2 14434.596} C_VEL
LIN {X 0,Y 296.797,Z 354.105,A -85,B 0,C 180,E1 14432.502,E2 14432.502} C_VEL
LIN {X 0,Y 295.354,Z 351.3,A -85,B 0,C 180,E1 14431.195,E2 14431.195} C_VEL
LIN {X 0,Y 293.337,Z 347.235,A -85,B 0,C 180,E1 14429.172,E2 14429.172} C_VEL
LIN {X 0,Y 291.114,Z 342.876,A -85,B 0,C 180,E1 14426.74,E2 14426.74} C_VEL
LIN {X 0,Y 288.896,Z 338.832,A -85,B 0,C 180,E1 14424.104,E2 14424.104} C_VEL
LIN {X 0,Y 287.834,Z 337.317,A -85,B 0,C 180,E1 14422.896,E2 14422.896} C_VEL
LIN {X 0,Y 285.304,Z 332.559,A -85,B 0,C 180,E1 14419.022,E2 14419.022} C_VEL
LIN {X 0,Y 282.392,Z 327.522,A -85,B 0,C 180,E1 14412.474,E2 14412.474} C_VEL
LIN {X 0,Y 282.37,Z 327.274,A -85,B 0,C 180,E1 14407.938,E2 14407.938} C_VEL
LIN {X 0,Y 282.37,Z 327.272,A -85,B 0,C 180,E1 14403.452,E2 14403.452} C_VEL
LIN {X 0,Y 282.348,Z 327.285,A -85,B 0,C 180,E1 14398.783,E2 14398.783} C_VEL
LIN {X 0,Y 282.425,Z 327.72,A -85,B 0,C 180,E1 14395.94,E2 14395.94} C_VEL
LIN {X 0,Y 285.978,Z 333.412,A -85,B 0,C 180,E1 14389.118,E2 14389.118} C_VEL
LIN {X 0,Y 288.041,Z 337.427,A -85,B 0,C 180,E1 14386.142,E2 14386.142} C_VEL
LIN {X 0,Y 289.259,Z 338.729,A -85,B 0,C 180,E1 14384.975,E2 14384.975} C_VEL
LIN {X 0,Y 291.325,Z 342.844,A -85,B 0,C 180,E1 14382.573,E2 14382.573} C_VEL
LIN {X 0,Y 292.38,Z 344.211,A -85,B 0,C 180,E1 14381.663,E2 14381.663} C_VEL
LIN {X 0,Y 294.621,Z 348.323,A -85,B 0,C 180,E1 14379.54,E2 14379.54} C_VEL
LIN {X 0,Y 298.029,Z 354.529,A -85,B 0,C 180,E1 14376.68,E2 14376.68} C_VEL
LIN {X 0,Y 300.849,Z 360.107,A -85,B 0,C 180,E1 14374.403,E2 14374.403} C_VEL
LIN {X 0,Y 304.889,Z 367.816,A -85,B 0,C 180,E1 14371.608,E2 14371.608} C_VEL
LIN {X 0,Y 307.814,Z 373.49,A -85,B 0,C 180,E1 14369.878,E2 14369.878} C_VEL
LIN {X 0,Y 316.729,Z 386.607,A -85,B 0,C 180,E1 14367.006,E2 14367.006} C_VEL
LIN {X 0,Y 326.956,Z 403.512,A -85,B 0,C 180,E1 14364.045,E2 14364.045} C_VEL
LIN {X 0,Y 335.325,Z 418.783,A -85,B 0,C 180,E1 14361.832,E2 14361.832} C_VEL
LIN {X 0,Y 336.697,Z 421.898,A -85,B 0,C 180,E1 14361.467,E2 14361.467} C_VEL
LIN {X 0,Y 337.37,Z 437.814,A -85,B 0,C 180,E1 14360.815,E2 14360.815} C_VEL
LIN {X 0,Y 326.808,Z 625.648,A -85,B 0,C 180,E1 14356.582,E2 14356.582} C_VEL
LIN {X 0,Y 324.311,Z 647.5,A -85,B 0,C 180,E1 14355.82,E2 14355.82} C_VEL
LIN {X 0,Y 320.735,Z 668.625,A -85,B 0,C 180,E1 14354.79,E2 14354.79} C_VEL
LIN {X 0,Y 316.617,Z 688.2,A -85,B 0,C 180,E1 14353.504,E2 14353.504} C_VEL
LIN {X 0,Y 312.082,Z 706.941,A -85,B 0,C 180,E1 14351.911,E2 14351.911} C_VEL
LIN {X 0,Y 307.269,Z 724.938,A -85,B 0,C 180,E1 14349.99,E2 14349.99} C_VEL
LIN {X 0,Y 302.301,Z 742.128,A -85,B 0,C 180,E1 14347.725,E2 14347.725} C_VEL
LIN {X 0,Y 297.403,Z 758.44,A -85,B 0,C 180,E1 14345.091,E2 14345.091} C_VEL
LIN {X 0,Y 292.89,Z 773.386,A -85,B 0,C 180,E1 14342.155,E2 14342.155} C_VEL
LIN {X 0,Y 288.865,Z 787.179,A -85,B 0,C 180,E1 14338.871,E2 14338.871} C_VEL
LIN {X 0,Y 285.571,Z 799.569,A -85,B 0,C 180,E1 14335.286,E2 14335.286} C_VEL
LIN {X 0,Y 283.203,Z 810.188,A -85,B 0,C 180,E1 14331.541,E2 14331.541} C_VEL
LIN {X 0,Y 281.699,Z 819.314,A -85,B 0,C 180,E1 14327.559,E2 14327.559} C_VEL
LIN {X 0,Y 281.093,Z 826.462,A -85,B 0,C 180,E1 14323.577,E2 14323.577} C_VEL
LIN {X 0,Y 281.142,Z 831.527,A -85,B 0,C 180,E1 14319.829,E2 14319.829} C_VEL
LIN {X 0,Y 281.522,Z 835.086,A -85,B 0,C 180,E1 14316.042,E2 14316.042} C_VEL
LIN {X 0,Y 281.873,Z 836.875,A -85,B 0,C 180,E1 14312.643,E2 14312.643} C_VEL
LIN {X 0,Y 281.975,Z 837.239,A -85,B 0,C 180,E1 14309.187,E2 14309.187} C_VEL
LIN {X 0,Y 281.742,Z 836.292,A -85,B 0,C 180,E1 14305.93,E2 14305.93} C_VEL
LIN {X 0,Y 281.325,Z 833.649,A -85,B 0,C 180,E1 14302.238,E2 14302.238} C_VEL
LIN {X 0,Y 281.058,Z 829.466,A -85,B 0,C 180,E1 14298.509,E2 14298.509} C_VEL
LIN {X 0,Y 281.291,Z 823.301,A -85,B 0,C 180,E1 14294.539,E2 14294.539} C_VEL
LIN {X 0,Y 282.363,Z 814.738,A -85,B 0,C 180,E1 14290.343,E2 14290.343} C_VEL
LIN {X 0,Y 284.388,Z 804.51,A -85,B 0,C 180,E1 14286.372,E2 14286.372} C_VEL
LIN {X 0,Y 287.337,Z 792.719,A -85,B 0,C 180,E1 14282.657,E2 14282.657} C_VEL
LIN {X 0,Y 290.825,Z 780.243,A -85,B 0,C 180,E1 14279.415,E2 14279.415} C_VEL
LIN {X 0,Y 295.211,Z 765.576,A -85,B 0,C 180,E1 14276.259,E2 14276.259} C_VEL
LIN {X 0,Y 300.035,Z 749.561,A -85,B 0,C 180,E1 14273.429,E2 14273.429} C_VEL
LIN {X 0,Y 305.177,Z 732.071,A -85,B 0,C 180,E1 14270.912,E2 14270.912} C_VEL
LIN {X 0,Y 310.209,Z 713.871,A -85,B 0,C 180,E1 14268.801,E2 14268.801} C_VEL
LIN {X 0,Y 314.895,Z 695.229,A -85,B 0,C 180,E1 14267.073,E2 14267.073} C_VEL
LIN {X 0,Y 319.137,Z 676.11,A -85,B 0,C 180,E1 14265.682,E2 14265.682} C_VEL
LIN {X 0,Y 322.871,Z 656.173,A -85,B 0,C 180,E1 14264.583,E2 14264.583} C_VEL
LIN {X 0,Y 325.768,Z 635.332,A -85,B 0,C 180,E1 14263.739,E2 14263.739} C_VEL
LIN {X 0,Y 327.543,Z 613.548,A -85,B 0,C 180,E1 14263.127,E2 14263.127} C_VEL
LIN {X 0,Y 337.322,Z 435.507,A -85,B 0,C 180,E1 14259.136,E2 14259.136} C_VEL
LIN {X 0,Y 336.383,Z 420.964,A -85,B 0,C 180,E1 14258.487,E2 14258.487} C_VEL
LIN {X 0,Y 327.352,Z 404.292,A -85,B 0,C 180,E1 14256.121,E2 14256.121} C_VEL
LIN {X 0,Y 318.165,Z 389.152,A -85,B 0,C 180,E1 14253.498,E2 14253.498} C_VEL
LIN {X 0,Y 310.074,Z 376.877,A -85,B 0,C 180,E1 14250.952,E2 14250.952} C_VEL
LIN {X 0,Y 307.079,Z 372.3,A -85,B 0,C 180,E1 14249.879,E2 14249.879} C_VEL
LIN {X 0,Y 302.151,Z 362.338,A -85,B 0,C 180,E1 14246.534,E2 14246.534} C_VEL
LIN {X 0,Y 299.009,Z 356.684,A -85,B 0,C 180,E1 14244.286,E2 14244.286} C_VEL
LIN {X 0,Y 297.215,Z 353.057,A -85,B 0,C 180,E1 14242.76,E2 14242.76} C_VEL
LIN {X 0,Y 294.739,Z 348.474,A -85,B 0,C 180,E1 14240.659,E2 14240.659} C_VEL
LIN {X 0,Y 292.419,Z 344.428,A -85,B 0,C 180,E1 14238.541,E2 14238.541} C_VEL
LIN {X 0,Y 291.573,Z 343.125,A -85,B 0,C 180,E1 14237.77,E2 14237.77} C_VEL
LIN {X 0,Y 289.394,Z 339.263,A -85,B 0,C 180,E1 14235.428,E2 14235.428} C_VEL
LIN {X 0,Y 288.505,Z 337.874,A -85,B 0,C 180,E1 14234.449,E2 14234.449} C_VEL
LIN {X 0,Y 286.26,Z 334.378,A -85,B 0,C 180,E1 14231.688,E2 14231.688} C_VEL
LIN {X 0,Y 285.578,Z 332.765,A -85,B 0,C 180,E1 14230.489,E2 14230.489} C_VEL
LIN {X 0,Y 282.527,Z 328.2,A -85,B 0,C 180,E1 14225.075,E2 14225.075} C_VEL
LIN {X 0,Y 282.365,Z 327.333,A -85,B 0,C 180,E1 14223.044,E2 14223.044} C_VEL
LIN {X 0,Y 282.372,Z 327.28,A -85,B 0,C 180,E1 14218.376,E2 14218.376} C_VEL
LIN {X 0,Y 282.353,Z 327.303,A -85,B 0,C 180,E1 14213.697,E2 14213.697} C_VEL
LIN {X 0,Y 282.363,Z 327.302,A -85,B 0,C 180,E1 14208.976,E2 14208.976} C_VEL
LIN {X 0,Y 282.488,Z 327.887,A -85,B 0,C 180,E1 14206.281,E2 14206.281} C_VEL
LIN {X 0,Y 285.785,Z 333.296,A -85,B 0,C 180,E1 14199.948,E2 14199.948} C_VEL
LIN {X 0,Y 287.795,Z 337.273,A -85,B 0,C 180,E1 14196.884,E2 14196.884} C_VEL
LIN {X 0,Y 288.847,Z 338.8,A -85,B 0,C 180,E1 14195.674,E2 14195.674} C_VEL
LIN {X 0,Y 291.137,Z 342.896,A -85,B 0,C 180,E1 14193.042,E2 14193.042} C_VEL
LIN {X 0,Y 294.191,Z 348.88,A -85,B 0,C 180,E1 14189.801,E2 14189.801} C_VEL
LIN {X 0,Y 296.717,Z 353.988,A -85,B 0,C 180,E1 14187.373,E2 14187.373} C_VEL
LIN {X 0,Y 303.78,Z 363.041,A -85,B 0,C 180,E1 14184.599,E2 14184.599} C_VEL
LIN {X 0,Y 311.069,Z 372.839,A -85,B 0,C 180,E1 14182.126,E2 14182.126} C_VEL
LIN {X 0,Y 320.552,Z 386.489,A -85,B 0,C 180,E1 14179.255,E2 14179.255} C_VEL
LIN {X 0,Y 329.948,Z 401.664,A -85,B 0,C 180,E1 14176.685,E2 14176.685} C_VEL
LIN {X 0,Y 336.894,Z 414.244,A -85,B 0,C 180,E1 14174.919,E2 14174.919} C_VEL
LIN {X 0,Y 329.698,Z 570.058,A -85,B 0,C 180,E1 14171.71,E2 14171.71} C_VEL
LIN {X 0,Y 328.353,Z 589.399,A -85,B 0,C 180,E1 14171.039,E2 14171.039} C_VEL
LIN {X 0,Y 326.214,Z 607.713,A -85,B 0,C 180,E1 14170.121,E2 14170.121} C_VEL
LIN {X 0,Y 323.267,Z 625.951,A -85,B 0,C 180,E1 14168.892,E2 14168.892} C_VEL
LIN {X 0,Y 319.625,Z 643.544,A -85,B 0,C 180,E1 14167.363,E2 14167.363} C_VEL
LIN {X 0,Y 315.485,Z 660.029,A -85,B 0,C 180,E1 14165.559,E2 14165.559} C_VEL
LIN {X 0,Y 311.009,Z 675.445,A -85,B 0,C 180,E1 14163.459,E2 14163.459} C_VEL
LIN {X 0,Y 306.307,Z 689.782,A -85,B 0,C 180,E1 14161.047,E2 14161.047} C_VEL
LIN {X 0,Y 301.577,Z 702.968,A -85,B 0,C 180,E1 14158.3,E2 14158.3} C_VEL
LIN {X 0,Y 297.104,Z 714.574,A -85,B 0,C 180,E1 14155.302,E2 14155.302} C_VEL
LIN {X 0,Y 293.064,Z 724.662,A -85,B 0,C 180,E1 14152.042,E2 14152.042} C_VEL
LIN {X 0,Y 289.568,Z 733.237,A -85,B 0,C 180,E1 14148.522,E2 14148.522} C_VEL
LIN {X 0,Y 286.735,Z 740.271,A -85,B 0,C 180,E1 14144.747,E2 14144.747} C_VEL
LIN {X 0,Y 284.752,Z 745.464,A -85,B 0,C 180,E1 14140.93,E2 14140.93} C_VEL
LIN {X 0,Y 283.422,Z 749.138,A -85,B 0,C 180,E1 14136.889,E2 14136.889} C_VEL
LIN {X 0,Y 282.774,Z 751.104,A -85,B 0,C 180,E1 14132.837,E2 14132.837} C_VEL
LIN {X 0,Y 282.67,Z 751.448,A -85,B 0,C 180,E1 14128.784,E2 14128.784} C_VEL
LIN {X 0,Y 283.077,Z 750.186,A -85,B 0,C 180,E1 14124.731,E2 14124.731} C_VEL
LIN {X 0,Y 284.105,Z 747.258,A -85,B 0,C 180,E1 14120.684,E2 14120.684} C_VEL
LIN {X 0,Y 285.762,Z 742.827,A -85,B 0,C 180,E1 14116.855,E2 14116.855} C_VEL
LIN {X 0,Y 288.21,Z 736.649,A -85,B 0,C 180,E1 14113.058,E2 14113.058} C_VEL
LIN {X 0,Y 291.35,Z 728.993,A -85,B 0,C 180,E1 14109.511,E2 14109.511} C_VEL
LIN {X 0,Y 295.262,Z 719.327,A -85,B 0,C 180,E1 14106.024,E2 14106.024} C_VEL
LIN {X 0,Y 299.443,Z 708.736,A -85,B 0,C 180,E1 14102.993,E2 14102.993} C_VEL
LIN {X 0,Y 303.928,Z 696.742,A -85,B 0,C 180,E1 14100.215,E2 14100.215} C_VEL
LIN {X 0,Y 308.75,Z 682.744,A -85,B 0,C 180,E1 14097.592,E2 14097.592} C_VEL
LIN {X 0,Y 313.468,Z 667.529,A -85,B 0,C 180,E1 14095.296,E2 14095.296} C_VEL
LIN {X 0,Y 317.791,Z 651.539,A -85,B 0,C 180,E1 14093.351,E2 14093.351} C_VEL
LIN {X 0,Y 321.723,Z 634.368,A -85,B 0,C 180,E1 14091.684,E2 14091.684} C_VEL
LIN {X 0,Y 324.984,Z 616.61,A -85,B 0,C 180,E1 14090.329,E2 14090.329} C_VEL
LIN {X 0,Y 327.594,Z 597.614,A -85,B 0,C 180,E1 14089.229,E2 14089.229} C_VEL
LIN {X 0,Y 329.331,Z 578.244,A -85,B 0,C 180,E1 14088.429,E2 14088.429} C_VEL
LIN {X 0,Y 330.034,Z 564.642,A -85,B 0,C 180,E1 14088.039,E2 14088.039} C_VEL
LIN {X 0,Y 329.643,Z 557.081,A -85,B 0,C 180,E1 14087.734,E2 14087.734} C_VEL
LIN {X 0,Y 326.126,Z 537.276,A -85,B 0,C 180,E1 14086.549,E2 14086.549} C_VEL
